LIN {X 0,Y 537.563,Z 430.245,A -85,B 0,C 180,E1 25559.467,E2 25559.467} C_VEL
LIN {X 0,Y 537.611,Z 430.26,A -85,B 0,C 180,E1 25556.268,E2 25556.268} C_VEL
LIN {X 0,Y 537.564,Z 430.265,A -85,B 0,C 180,E1 25552.948,E2 25552.948} C_VEL
LIN {X 0,Y 537.598,Z 430.246,A -85,B 0,C 180,E1 25549.606,E2 25549.606} C_VEL
LIN {X 0,Y 537.598,Z 430.246,A -85,B 0,C 180,E1 25546.337,E2 25546.337} C_VEL
LIN {X 0,Y 537.576,Z 430.262,A -85,B 0,C 180,E1 25542.949,E2 25542.949} C_VEL
LIN {X 0,Y 537.624,Z 430.26,A -85,B 0,C 180,E1 25539.613,E2 25539.613} C_VEL
LIN {X 0,Y 537.599,Z 430.262,A -85,B 0,C 180,E1 25536.313,E2 25536.313} C_VEL
LIN {X 0,Y 537.589,Z 430.264,A -85,B 0,C 180,E1 25532.891,E2 25532.891} C_VEL
LIN {X 0,Y 537.63,Z 430.257,A -85,B 0,C 180,E1 25529.611,E2 25529.611} C_VEL
LIN {X 0,Y 537.595,Z 430.198,A -85,B 0,C 180,E1 25526.212,E2 25526.212} C_VEL
LIN {X 0,Y 537.597,Z 430.248,A -85,B 0,C 180,E1 25522.755,E2 25522.755} C_VEL
LIN {X 0,Y 537.67,Z 430.675,A -85,B 0,C 180,E1 25522.164,E2 25522.164} C_VEL
LIN {X 0,Y 539.489,Z 434.5,A -85,B 0,C 180,E1 25521.457,E2 25521.457} C_VEL
LIN {X 0,Y 545.731,Z 448.172,A -85,B 0,C 180,E1 25519.149,E2 25519.149} C_VEL
LIN {X 0,Y 551.276,Z 460.441,A -85,B 0,C 180,E1 25517.249,E2 25517.249} C_VEL
LIN {X 0,Y 565.395,Z 481.878,A -85,B 0,C 180,E1 25515.423,E2 25515.423} C_VEL
LIN {X 0,Y 579.093,Z 504.577,A -85,B 0,C 180,E1 25513.764,E2 25513.764} C_VEL
LIN {X 0,Y 572.062,Z 749.764,A -85,B 0,C 180,E1 25510.284,E2 25510.284} C_VEL
LIN {X 0,Y 569.354,Z 843.896,A -85,B 0,C 180,E1 25508.929,E2 25508.929} C_VEL
LIN {X 0,Y 567.836,Z 869.316,A -85,B 0,C 180,E1 25508.396,E2 25508.396} C_VEL
LIN {X 0,Y 566.137,Z 891.39,A -85,B 0,C 180,E1 25507.777,E2 25507.777} C_VEL
LIN {X 0,Y 563.86,Z 915.912,A -85,B 0,C 180,E1 25506.893,E2 25506.893} C_VEL
LIN {X 0,Y 561.758,Z 935.486,A -85,B 0,C 180,E1 25506.034,E2 25506.034} C_VEL
LIN {X 0,Y 559.066,Z 958.281,A -85,B 0,C 180,E1 25504.85,E2 25504.85} C_VEL
LIN {X 0,Y 556.415,Z 978.46,A -85,B 0,C 180,E1 25503.607,E2 25503.607} C_VEL
LIN {X 0,Y 553.585,Z 999.25,A -85,B 0,C 180,E1 25502.13,E2 25502.13} C_VEL
LIN {X 0,Y 550.795,Z 1018.62,A -85,B 0,C 180,E1 25500.52,E2 25500.52} C_VEL
LIN {X 0,Y 548.082,Z 1037.54,A -85,B 0,C 180,E1 25498.732,E2 25498.732} C_VEL
LIN {X 0,Y 545.584,Z 1054.652,A -85,B 0,C 180,E1 25496.857,E2 25496.857} C_VEL
LIN {X 0,Y 543.312,Z 1071.181,A -85,B 0,C 180,E1 25494.81,E2 25494.81} C_VEL
LIN {X 0,Y 541.344,Z 1085.798,A -85,B 0,C 180,E1 25492.708,E2 25492.708} C_VEL
LIN {X 0,Y 539.711,Z 1099.37,A -85,B 0,C 180,E1 25490.497,E2 25490.497} C_VEL
LIN {X 0,Y 538.397,Z 1111.524,A -85,B 0,C 180,E1 25488.18,E2 25488.18} C_VEL
LIN {X 0,Y 537.464,Z 1121.5,A -85,B 0,C 180,E1 25485.982,E2 25485.982} C_VEL
LIN {X 0,Y 536.711,Z 1131.437,A -85,B 0,C 180,E1 25483.357,E2 25483.357} C_VEL
LIN {X 0,Y 536.314,Z 1137.908,A -85,B 0,C 180,E1 25481.285,E2 25481.285} C_VEL
LIN {X 0,Y 536.061,Z 1144.005,A -85,B 0,C 180,E1 25478.906,E2 25478.906} C_VEL
LIN {X 0,Y 535.956,Z 1148.651,A -85,B 0,C 180,E1 25476.427,E2 25476.427} C_VEL
LIN {X 0,Y 535.926,Z 1151.599,A -85,B 0,C 180,E1 25474.173,E2 25474.173} C_VEL
LIN {X 0,Y 535.906,Z 1153.482,A -85,B 0,C 180,E1 25471.604,E2 25471.604} C_VEL
LIN {X 0,Y 535.895,Z 1153.67,A -85,B 0,C 180,E1 25469.252,E2 25469.252} C_VEL
LIN {X 0,Y 535.893,Z 1152.72,A -85,B 0,C 180,E1 25467.112,E2 25467.112} C_VEL
LIN {X 0,Y 535.911,Z 1150.294,A -85,B 0,C 180,E1 25464.647,E2 25464.647} C_VEL
LIN {X 0,Y 535.982,Z 1146.4,A -85,B 0,C 180,E1 25462.281,E2 25462.281} C_VEL
LIN {X 0,Y 536.155,Z 1141.661,A -85,B 0,C 180,E1 25460.121,E2 25460.121} C_VEL
LIN {X 0,Y 536.527,Z 1134.357,A -85,B 0,C 180,E1 25457.515,E2 25457.515} C_VEL
LIN {X 0,Y 537.075,Z 1126.302,A -85,B 0,C 180,E1 25455.223,E2 25455.223} C_VEL
LIN {X 0,Y 537.942,Z 1116.295,A -85,B 0,C 180,E1 25452.81,E2 25452.81} C_VEL
LIN {X 0,Y 539.101,Z 1104.77,A -85,B 0,C 180,E1 25450.497,E2 25450.497} C_VEL
LIN {X 0,Y 540.565,Z 1092.172,A -85,B 0,C 180,E1 25448.288,E2 25448.288} C_VEL
LIN {X 0,Y 542.432,Z 1077.521,A -85,B 0,C 180,E1 25446.075,E2 25446.075} C_VEL
LIN {X 0,Y 544.396,Z 1063.086,A -85,B 0,C 180,E1 25444.156,E2 25444.156} C_VEL
LIN {X 0,Y 547.004,Z 1044.796,A -85,B 0,C 180,E1 25442.039,E2 25442.039} C_VEL
LIN {X 0,Y 549.352,Z 1028.487,A -85,B 0,C 180,E1 25440.385,E2 25440.385} C_VEL
LIN {X 0,Y 552.424,Z 1007.258,A -85,B 0,C 180,E1 25438.515,E2 25438.515} C_VEL
LIN {X 0,Y 554.922,Z 989.488,A -85,B 0,C 180,E1 25437.155,E2 25437.155} C_VEL
LIN {X 0,Y 557.868,Z 967.473,A -85,B 0,C 180,E1 25435.695,E2 25435.695} C_VEL
LIN {X 0,Y 560.34,Z 947.273,A -85,B 0,C 180,E1 25434.553,E2 25434.553} C_VEL
LIN {X 0,Y 563.059,Z 923.705,A -85,B 0,C 180,E1 25433.431,E2 25433.431} C_VEL
LIN {X 0,Y 565.125,Z 902.488,A -85,B 0,C 180,E1 25432.602,E2 25432.602} C_VEL
LIN {X 0,Y 567.194,Z 878.756,A -85,B 0,C 180,E1 25431.848,E2 25431.848} C_VEL
LIN {X 0,Y 568.742,Z 855.353,A -85,B 0,C 180,E1 25431.295,E2 25431.295} C_VEL
LIN {X 0,Y 569.818,Z 831.659,A -85,B 0,C 180,E1 25430.878,E2 25430.878} C_VEL
LIN {X 0,Y 576.437,Z 593.145,A -85,B 0,C 180,E1 25427.493,E2 25427.493} C_VEL
LIN {X 0,Y 578.891,Z 504.261,A -85,B 0,C 180,E1 25426.219,E2 25426.219} C_VEL
LIN {X 0,Y 564.561,Z 480.573,A -85,B 0,C 180,E1 25424.483,E2 25424.483} C_VEL
LIN {X 0,Y 551.107,Z 460.145,A -85,B 0,C 180,E1 25422.732,E2 25422.732} C_VEL
LIN {X 0,Y 544.782,Z 446.05,A -85,B 0,C 180,E1 25420.521,E2 25420.521} C_VEL
LIN {X 0,Y 539.013,Z 433.83,A -85,B 0,C 180,E1 25418.421,E2 25418.421} C_VEL
LIN {X 0,Y 537.627,Z 430.435,A -85,B 0,C 180,E1 25417.774,E2 25417.774} C_VEL
LIN {X 0,Y 537.619,Z 430.197,A -85,B 0,C 180,E1 25414.43,E2 25414.43} C_VEL
LIN {X 0,Y 537.596,Z 430.267,A -85,B 0,C 180,E1 25411.135,E2 25411.135} C_VEL
LIN {X 0,Y 537.604,Z 430.267,A -85,B 0,C 180,E1 25407.709,E2 25407.709} C_VEL
LIN {X 0,Y 537.629,Z 430.259,A -85,B 0,C 180,E1 25404.312,E2 25404.312} C_VEL
LIN {X 0,Y 537.586,Z 430.261,A -85,B 0,C 180,E1 25400.98,E2 25400.98} C_VEL
LIN {X 0,Y 537.59,Z 430.25,A -85,B 0,C 180,E1 25397.536,E2 25397.536} C_VEL
LIN {X 0,Y 537.633,Z 430.239,A -85,B 0,C 180,E1 25394.211,E2 25394.211} C_VEL
LIN {X 0,Y 537.573,Z 430.257,A -85,B 0,C 180,E1 25390.86,E2 25390.86} C_VEL
LIN {X 0,Y 537.591,Z 430.266,A -85,B 0,C 180,E1 25387.481,E2 25387.481} C_VEL
LIN {X 0,Y 537.597,Z 430.253,A -85,B 0,C 180,E1 25384.267,E2 25384.267} C_VEL
LIN {X 0,Y 537.56,Z 430.244,A -85,B 0,C 180,E1 25380.959,E2 25380.959} C_VEL
LIN {X 0,Y 537.618,Z 430.255,A -85,B 0,C 180,E1 25377.762,E2 25377.762} C_VEL
LIN {X 0,Y 537.561,Z 430.266,A -85,B 0,C 180,E1 25374.449,E2 25374.449} C_VEL
LIN {X 0,Y 537.558,Z 430.254,A -85,B 0,C 180,E1 25371.003,E2 25371.003} C_VEL
LIN {X 0,Y 537.604,Z 430.244,A -85,B 0,C 180,E1 25367.759,E2 25367.759} C_VEL
LIN {X 0,Y 537.545,Z 430.267,A -85,B 0,C 180,E1 25364.574,E2 25364.574} C_VEL
LIN {X 0,Y 537.598,Z 430.266,A -85,B 0,C 180,E1 25361.343,E2 25361.343} C_VEL
LIN {X 0,Y 537.544,Z 430.262,A -85,B 0,C 180,E1 25358.156,E2 25358.156} C_VEL
LIN {X 0,Y 537.539,Z 430.259,A -85,B 0,C 180,E1 25354.67,E2 25354.67} C_VEL
LIN {X 0,Y 537.604,Z 430.249,A -85,B 0,C 180,E1 25351.387,E2 25351.387} C_VEL
LIN {X 0,Y 537.524,Z 430.258,A -85,B 0,C 180,E1 25348.223,E2 25348.223} C_VEL
LIN {X 0,Y 537.558,Z 430.212,A -85,B 0,C 180,E1 25344.917,E2 25344.917} C_VEL
LIN {X 0,Y 537.544,Z 430.254,A -85,B 0,C 180,E1 25341.718,E2 25341.718} C_VEL
LIN {X 0,Y 537.659,Z 430.659,A -85,B 0,C 180,E1 25341.25,E2 25341.25} C_VEL
LIN {X 0,Y 539.072,Z 434.068,A -85,B 0,C 180,E1 25340.628,E2 25340.628} C_VEL
LIN {X 0,Y 543.735,Z 444.332,A -85,B 0,C 180,E1 25338.827,E2 25338.827} C_VEL
LIN {X 0,Y 548.585,Z 455.234,A -85,B 0,C 180,E1 25337.025,E2 25337.025} C_VEL
LIN {X 0,Y 555.423,Z 471.599,A -85,B 0,C 180,E1 25334.529,E2 25334.529} C_VEL
LIN {X 0,Y 562.151,Z 489.574,A -85,B 0,C 180,E1 25332.046,E2 25332.046} C_VEL
LIN {X 0,Y 563.644,Z 493.192,A -85,B 0,C 180,E1 25331.625,E2 25331.625} C_VEL
LIN {X 0,Y 567.174,Z 499.748,A -85,B 0,C 180,E1 25331.178,E2 25331.178} C_VEL
LIN {X 0,Y 575.924,Z 543.536,A -85,B 0,C 180,E1 25329.673,E2 25329.673} C_VEL
LIN {X 0,Y 570.099,Z 791.217,A -85,B 0,C 180,E1 25326.365,E2 25326.365} C_VEL
LIN {X 0,Y 569.15,Z 798.915,A -85,B 0,C 180,E1 25326.325,E2 25326.325} C_VEL
LIN {X 0,Y 563.752,Z 819.438,A -85,B 0,C 180,E1 25326.446,E2 25326.446} C_VEL
LIN {X 0,Y 563.016,Z 826.045,A -85,B 0,C 180,E1 25326.405,E2 25326.405} C_VEL
LIN {X 0,Y 561.954,Z 855.614,A -85,B 0,C 180,E1 25325.948,E2 25325.948} C_VEL
LIN {X 0,Y 560.633,Z 876.398,A -85,B 0,C 180,E1 25325.48,E2 25325.48} C_VEL
LIN {X 0,Y 558.691,Z 899.351,A -85,B 0,C 180,E1 25324.782,E2 25324.782} C_VEL
LIN {X 0,Y 556.656,Z 919.096,A -85,B 0,C 180,E1 25324.024,E2 25324.024} C_VEL
LIN {X 0,Y 553.94,Z 941.342,A -85,B 0,C 180,E1 25322.972,E2 25322.972} C_VEL
LIN {X 0,Y 551.282,Z 960.921,A -85,B 0,C 180,E1 25321.857,E2 25321.857} C_VEL
LIN {X 0,Y 548.337,Z 980.641,A -85,B 0,C 180,E1 25320.521,E2 25320.521} C_VEL
LIN {X 0,Y 545.53,Z 998.333,A -85,B 0,C 180,E1 25319.127,E2 25319.127} C_VEL
LIN {X 0,Y 542.444,Z 1016.652,A -85,B 0,C 180,E1 25317.441,E2 25317.441} C_VEL
LIN {X 0,Y 539.637,Z 1033.467,A -85,B 0,C 180,E1 25315.651,E2 25315.651} C_VEL
LIN {X 0,Y 536.965,Z 1048.953,A -85,B 0,C 180,E1 25313.717,E2 25313.717} C_VEL
LIN {X 0,Y 534.607,Z 1063.539,A -85,B 0,C 180,E1 25311.62,E2 25311.62} C_VEL
LIN {X 0,Y 532.672,Z 1075.997,A -85,B 0,C 180,E1 25309.52,E2 25309.52} C_VEL
LIN {X 0,Y 530.943,Z 1088.34,A -85,B 0,C 180,E1 25307.085,E2 25307.085} C_VEL
LIN {X 0,Y 529.803,Z 1097.772,A -85,B 0,C 180,E1 25304.873,E2 25304.873} C_VEL
LIN {X 0,Y 528.907,Z 1106.716,A -85,B 0,C 180,E1 25302.335,E2 25302.335} C_VEL
LIN {X 0,Y 528.402,Z 1113.315,A -85,B 0,C 180,E1 25300.026,E2 25300.026} C_VEL
LIN {X 0,Y 528.103,Z 1118.824,A -85,B 0,C 180,E1 25297.507,E2 25297.507} C_VEL
LIN {X 0,Y 527.976,Z 1122.478,A -85,B 0,C 180,E1 25295.216,E2 25295.216} C_VEL
LIN {X 0,Y 527.922,Z 1124.991,A -85,B 0,C 180,E1 25292.605,E2 25292.605} C_VEL
LIN {X 0,Y 527.918,Z 1125.857,A -85,B 0,C 180,E1 25290.326,E2 25290.326} C_VEL
LIN {X 0,Y 527.922,Z 1125.244,A -85,B 0,C 180,E1 25287.72,E2 25287.72} C_VEL
LIN {X 0,Y 527.946,Z 1123.366,A -85,B 0,C 180,E1 25285.438,E2 25285.438} C_VEL
LIN {X 0,Y 528.064,Z 1119.589,A -85,B 0,C 180,E1 25282.821,E2 25282.821} C_VEL
LIN {X 0,Y 528.304,Z 1114.866,A -85,B 0,C 180,E1 25280.522,E2 25280.522} C_VEL
LIN {X 0,Y 528.798,Z 1108.023,A -85,B 0,C 180,E1 25277.995,E2 25277.995} C_VEL
LIN {X 0,Y 529.546,Z 1100.239,A -85,B 0,C 180,E1 25275.679,E2 25275.679} C_VEL
LIN {X 0,Y 530.706,Z 1090.239,A -85,B 0,C 180,E1 25273.246,E2 25273.246} C_VEL
LIN {X 0,Y 532.27,Z 1078.959,A -85,B 0,C 180,E1 25270.921,E2 25270.921} C_VEL
LIN {X 0,Y 534.178,Z 1066.132,A -85,B 0,C 180,E1 25268.707,E2 25268.707} C_VEL
LIN {X 0,Y 536.604,Z 1051.259,A -85,B 0,C 180,E1 25266.499,E2 25266.499} C_VEL
LIN {X 0,Y 539.08,Z 1036.58,A -85,B 0,C 180,E1 25264.63,E2 25264.63} C_VEL
LIN {X 0,Y 542.044,Z 1019.136,A -85,B 0,C 180,E1 25262.716,E2 25262.716} C_VEL
LIN {X 0,Y 544.839,Z 1002.518,A -85,B 0,C 180,E1 25261.141,E2 25261.141} C_VEL
LIN {X 0,Y 547.91,Z 983.484,A -85,B 0,C 180,E1 25259.597,E2 25259.597} C_VEL
LIN {X 0,Y 550.709,Z 965.137,A -85,B 0,C 180,E1 25258.317,E2 25258.317} C_VEL
LIN {X 0,Y 553.497,Z 944.852,A -85,B 0,C 180,E1 25257.122,E2 25257.122} C_VEL
LIN {X 0,Y 556.047,Z 924.615,A -85,B 0,C 180,E1 25256.12,E2 25256.12} C_VEL
LIN {X 0,Y 558.333,Z 903.1,A -85,B 0,C 180,E1 25255.256,E2 25255.256} C_VEL
LIN {X 0,Y 560.263,Z 881.795,A -85,B 0,C 180,E1 25254.571,E2 25254.571} C_VEL
LIN {X 0,Y 561.795,Z 858.909,A -85,B 0,C 180,E1 25254.024,E2 25254.024} C_VEL
LIN {X 0,Y 562.808,Z 836.018,A -85,B 0,C 180,E1 25253.636,E2 25253.636} C_VEL
LIN {X 0,Y 568.803,Z 586.916,A -85,B 0,C 180,E1 25250.287,E2 25250.287} C_VEL
LIN {X 0,Y 569.81,Z 544.081,A -85,B 0,C 180,E1 25249.691,E2 25249.691} C_VEL
LIN {X 0,Y 561.524,Z 502.952,A -85,B 0,C 180,E1 25248.235,E2 25248.235} C_VEL
LIN {X 0,Y 554.808,Z 491.423,A -85,B 0,C 180,E1 25247.334,E2 25247.334} C_VEL
LIN {X 0,Y 547.67,Z 472.631,A -85,B 0,C 180,E1 25244.66,E2 25244.66} C_VEL
LIN {X 0,Y 540.405,Z 455.19,A -85,B 0,C 180,E1 25241.909,E2 25241.909} C_VEL
LIN {X 0,Y 534.741,Z 442.856,A -85,B 0,C 180,E1 25239.754,E2 25239.754} C_VEL
LIN {X 0,Y 531.038,Z 434.894,A -85,B 0,C 180,E1 25238.278,E2 25238.278} C_VEL
LIN {X 0,Y 529.624,Z 431.422,A -85,B 0,C 180,E1 25237.575,E2 25237.575} C_VEL
LIN {X 0,Y 529.637,Z 431.208,A -85,B 0,C 180,E1 25234.497,E2 25234.497} C_VEL
LIN {X 0,Y 529.602,Z 431.244,A -85,B 0,C 180,E1 25231.279,E2 25231.279} C_VEL
LIN {X 0,Y 529.59,Z 431.245,A -85,B 0,C 180,E1 25227.919,E2 25227.919} C_VEL
LIN {X 0,Y 529.649,Z 431.237,A -85,B 0,C 180,E1 25224.659,E2 25224.659} C_VEL
LIN {X 0,Y 529.592,Z 431.247,A -85,B 0,C 180,E1 25221.439,E2 25221.439} C_VEL
LIN {X 0,Y 529.637,Z 431.25,A -85,B 0,C 180,E1 25218.15,E2 25218.15} C_VEL
LIN {X 0,Y 529.613,Z 431.258,A -85,B 0,C 180,E1 25214.99,E2 25214.99} C_VEL
LIN {X 0,Y 529.607,Z 431.248,A -85,B 0,C 180,E1 25211.516,E2 25211.516} C_VEL
LIN {X 0,Y 529.676,Z 431.228,A -85,B 0,C 180,E1 25208.249,E2 25208.249} C_VEL
LIN {X 0,Y 529.617,Z 431.251,A -85,B 0,C 180,E1 25204.982,E2 25204.982} C_VEL
LIN {X 0,Y 529.625,Z 431.257,A -85,B 0,C 180,E1 25201.515,E2 25201.515} C_VEL
LIN {X 0,Y 529.662,Z 431.233,A -85,B 0,C 180,E1 25198.377,E2 25198.377} C_VEL
LIN {X 0,Y 529.621,Z 431.237,A -85,B 0,C 180,E1 25195.018,E2 25195.018} C_VEL
LIN {X 0,Y 529.661,Z 431.248,A -85,B 0,C 180,E1 25191.642,E2 25191.642} C_VEL
LIN {X 0,Y 529.66,Z 431.251,A -85,B 0,C 180,E1 25188.346,E2 25188.346} C_VEL
LIN {X 0,Y 529.634,Z 431.241,A -85,B 0,C 180,E1 25185.01,E2 25185.01} C_VEL
LIN {X 0,Y 529.685,Z 431.228,A -85,B 0,C 180,E1 25181.718,E2 25181.718} C_VEL
LIN {X 0,Y 529.653,Z 431.237,A -85,B 0,C 180,E1 25178.4,E2 25178.4} C_VEL
LIN {X 0,Y 529.651,Z 431.243,A -85,B 0,C 180,E1 25174.98,E2 25174.98} C_VEL
LIN {X 0,Y 529.696,Z 431.238,A -85,B 0,C 180,E1 25171.595,E2 25171.595} C_VEL
LIN {X 0,Y 529.663,Z 431.229,A -85,B 0,C 180,E1 25168.218,E2 25168.218} C_VEL
LIN {X 0,Y 529.65,Z 431.203,A -85,B 0,C 180,E1 25164.712,E2 25164.712} C_VEL
LIN {X 0,Y 529.728,Z 431.569,A -85,B 0,C 180,E1 25163.161,E2 25163.161} C_VEL
LIN {X 0,Y 531.079,Z 434.887,A -85,B 0,C 180,E1 25162.545,E2 25162.545} C_VEL
LIN {X 0,Y 534.312,Z 441.615,A -85,B 0,C 180,E1 25161.315,E2 25161.315} C_VEL
LIN {X 0,Y 539.492,Z 452.574,A -85,B 0,C 180,E1 25159.417,E2 25159.417} C_VEL
LIN {X 0,Y 543.297,Z 460.954,A -85,B 0,C 180,E1 25158.099,E2 25158.099} C_VEL
LIN {X 0,Y 557.37,Z 482.066,A -85,B 0,C 180,E1 25156.21,E2 25156.21} C_VEL
LIN {X 0,Y 571.534,Z 505.199,A -85,B 0,C 180,E1 25154.438,E2 25154.438} C_VEL
LIN {X 0,Y 573.043,Z 508.177,A -85,B 0,C 180,E1 25154.248,E2 25154.248} C_VEL
LIN {X 0,Y 565.685,Z 754.075,A -85,B 0,C 180,E1 25150.727,E2 25150.727} C_VEL
LIN {X 0,Y 562.975,Z 844.037,A -85,B 0,C 180,E1 25149.419,E2 25149.419} C_VEL
LIN {X 0,Y 561.402,Z 869.3,A -85,B 0,C 180,E1 25148.885,E2 25148.885} C_VEL
LIN {X 0,Y 559.62,Z 891.562,A -85,B 0,C 180,E1 25148.255,E2 25148.255} C_VEL
LIN {X 0,Y 557.329,Z 915.295,A -85,B 0,C 180,E1 25147.394,E2 25147.394} C_VEL
LIN {X 0,Y 555.015,Z 935.997,A -85,B 0,C 180,E1 25146.478,E2 25146.478} C_VEL
LIN {X 0,Y 552.089,Z 959.513,A -85,B 0,C 180,E1 25145.233,E2 25145.233} C_VEL
LIN {X 0,Y 549.449,Z 978.788,A -85,B 0,C 180,E1 25144.028,E2 25144.028} C_VEL
LIN {X 0,Y 546.495,Z 999.423,A -85,B 0,C 180,E1 25142.542,E2 25142.542} C_VEL
LIN {X 0,Y 543.614,Z 1018.503,A -85,B 0,C 180,E1 25140.937,E2 25140.937} C_VEL
LIN {X 0,Y 540.813,Z 1037.151,A -85,B 0,C 180,E1 25139.155,E2 25139.155} C_VEL
LIN {X 0,Y 538.096,Z 1054.746,A -85,B 0,C 180,E1 25137.201,E2 25137.201} C_VEL
LIN {X 0,Y 535.733,Z 1071.067,A -85,B 0,C 180,E1 25135.149,E2 25135.149} C_VEL
LIN {X 0,Y 533.588,Z 1086.161,A -85,B 0,C 180,E1 25132.94,E2 25132.94} C_VEL
LIN {X 0,Y 531.882,Z 1099.66,A -85,B 0,C 180,E1 25130.697,E2 25130.697} C_VEL
LIN {X 0,Y 530.496,Z 1111.691,A -85,B 0,C 180,E1 25128.347,E2 25128.347} C_VEL
LIN {X 0,Y 529.483,Z 1122.099,A -85,B 0,C 180,E1 25126.004,E2 25126.004} C_VEL
LIN {X 0,Y 528.734,Z 1131.506,A -85,B 0,C 180,E1 25123.451,E2 25123.451} C_VEL
LIN {X 0,Y 528.31,Z 1138.247,A -85,B 0,C 180,E1 25121.241,E2 25121.241} C_VEL
LIN {X 0,Y 528.052,Z 1144.655,A -85,B 0,C 180,E1 25118.603,E2 25118.603} C_VEL
LIN {X 0,Y 527.955,Z 1148.75,A -85,B 0,C 180,E1 25116.306,E2 25116.306} C_VEL
LIN {X 0,Y 527.925,Z 1151.615,A -85,B 0,C 180,E1 25114.018,E2 25114.018} C_VEL
LIN {X 0,Y 527.916,Z 1153.342,A -85,B 0,C 180,E1 25111.302,E2 25111.302} C_VEL
LIN {X 0,Y 527.902,Z 1153.437,A -85,B 0,C 180,E1 25109.132,E2 25109.132} C_VEL
LIN {X 0,Y 527.899,Z 1152.434,A -85,B 0,C 180,E1 25106.96,E2 25106.96} C_VEL
LIN {X 0,Y 527.927,Z 1149.742,A -85,B 0,C 180,E1 25104.348,E2 25104.348} C_VEL
LIN {X 0,Y 528,Z 1145.941,A -85,B 0,C 180,E1 25102.054,E2 25102.054} C_VEL
LIN {X 0,Y 528.189,Z 1140.872,A -85,B 0,C 180,E1 25099.75,E2 25099.75} C_VEL
LIN {X 0,Y 528.611,Z 1133.332,A -85,B 0,C 180,E1 25097.103,E2 25097.103} C_VEL
LIN {X 0,Y 529.183,Z 1125.554,A -85,B 0,C 180,E1 25094.885,E2 25094.885} C_VEL
LIN {X 0,Y 530.17,Z 1114.882,A -85,B 0,C 180,E1 25092.323,E2 25092.323} C_VEL
LIN {X 0,Y 531.368,Z 1103.818,A -85,B 0,C 180,E1 25090.087,E2 25090.087} C_VEL
LIN {X 0,Y 533.053,Z 1090.481,A -85,B 0,C 180,E1 25087.734,E2 25087.734} C_VEL
LIN {X 0,Y 535.015,Z 1075.841,A -85,B 0,C 180,E1 25085.527,E2 25085.527} C_VEL
LIN {X 0,Y 537.29,Z 1060.404,A -85,B 0,C 180,E1 25083.472,E2 25083.472} C_VEL
LIN {X 0,Y 539.885,Z 1042.843,A -85,B 0,C 180,E1 25081.456,E2 25081.456} C_VEL
LIN {X 0,Y 542.709,Z 1024.671,A -85,B 0,C 180,E1 25079.619,E2 25079.619} C_VEL
LIN {X 0,Y 545.521,Z 1005.807,A -85,B 0,C 180,E1 25077.979,E2 25077.979} C_VEL
LIN {X 0,Y 548.322,Z 986.768,A -85,B 0,C 180,E1 25076.521,E2 25076.521} C_VEL
LIN {X 0,Y 551.332,Z 964.918,A -85,B 0,C 180,E1 25075.091,E2 25075.091} C_VEL
LIN {X 0,Y 553.941,Z 944.652,A -85,B 0,C 180,E1 25073.953,E2 25073.953} C_VEL
LIN {X 0,Y 556.71,Z 921.019,A -85,B 0,C 180,E1 25072.847,E2 25072.847} C_VEL
LIN {X 0,Y 558.801,Z 900.349,A -85,B 0,C 180,E1 25072.046,E2 25072.046} C_VEL
LIN {X 0,Y 560.965,Z 875.428,A -85,B 0,C 180,E1 25071.276,E2 25071.276} C_VEL
LIN {X 0,Y 562.43,Z 853.769,A -85,B 0,C 180,E1 25070.772,E2 25070.772} C_VEL
LIN {X 0,Y 563.576,Z 827.693,A -85,B 0,C 180,E1 25070.327,E2 25070.327} C_VEL
LIN {X 0,Y 570.432,Z 591.297,A -85,B 0,C 180,E1 25066.942,E2 25066.942} C_VEL
LIN {X 0,Y 572.854,Z 507.561,A -85,B 0,C 180,E1 25065.731,E2 25065.731} C_VEL
LIN {X 0,Y 559.284,Z 485.093,A -85,B 0,C 180,E1 25064.046,E2 25064.046} C_VEL
LIN {X 0,Y 545.384,Z 464.099,A -85,B 0,C 180,E1 25062.216,E2 25062.216} C_VEL
LIN {X 0,Y 542.908,Z 460.138,A -85,B 0,C 180,E1 25061.814,E2 25061.814} C_VEL
LIN {X 0,Y 535.54,Z 443.92,A -85,B 0,C 180,E1 25059.129,E2 25059.129} C_VEL
LIN {X 0,Y 531.026,Z 434.81,A -85,B 0,C 180,E1 25057.459,E2 25057.459} C_VEL
LIN {X 0,Y 529.703,Z 431.4,A -85,B 0,C 180,E1 25056.796,E2 25056.796} C_VEL
LIN {X 0,Y 529.647,Z 431.187,A -85,B 0,C 180,E1 25053.443,E2 25053.443} C_VEL
LIN {X 0,Y 529.685,Z 431.239,A -85,B 0,C 180,E1 25050.016,E2 25050.016} C_VEL
LIN {X 0,Y 529.683,Z 431.239,A -85,B 0,C 180,E1 25046.576,E2 25046.576} C_VEL
LIN {X 0,Y 529.645,Z 431.246,A -85,B 0,C 180,E1 25043.163,E2 25043.163} C_VEL
LIN {X 0,Y 529.67,Z 431.247,A -85,B 0,C 180,E1 25039.75,E2 25039.75} C_VEL
LIN {X 0,Y 529.682,Z 431.249,A -85,B 0,C 180,E1 25036.336,E2 25036.336} C_VEL
LIN {X 0,Y 529.633,Z 431.247,A -85,B 0,C 180,E1 25033.054,E2 25033.054} C_VEL
LIN {X 0,Y 529.666,Z 431.231,A -85,B 0,C 180,E1 25029.672,E2 25029.672} C_VEL
LIN {X 0,Y 529.645,Z 431.245,A -85,B 0,C 180,E1 25026.504,E2 25026.504} C_VEL
LIN {X 0,Y 529.627,Z 431.257,A -85,B 0,C 180,E1 25023.03,E2 25023.03} C_VEL
LIN {X 0,Y 529.678,Z 431.237,A -85,B 0,C 180,E1 25019.676,E2 25019.676} C_VEL
LIN {X 0,Y 529.625,Z 431.232,A -85,B 0,C 180,E1 25016.428,E2 25016.428} C_VEL
LIN {X 0,Y 529.618,Z 431.247,A -85,B 0,C 180,E1 25012.951,E2 25012.951} C_VEL
LIN {X 0,Y 529.675,Z 431.253,A -85,B 0,C 180,E1 25009.669,E2 25009.669} C_VEL
LIN {X 0,Y 529.612,Z 431.249,A -85,B 0,C 180,E1 25006.35,E2 25006.35} C_VEL
LIN {X 0,Y 529.609,Z 431.24,A -85,B 0,C 180,E1 25002.809,E2 25002.809} C_VEL
LIN {X 0,Y 529.664,Z 431.235,A -85,B 0,C 180,E1 24999.559,E2 24999.559} C_VEL
LIN {X 0,Y 529.598,Z 431.252,A -85,B 0,C 180,E1 24996.305,E2 24996.305} C_VEL
LIN {X 0,Y 529.62,Z 431.253,A -85,B 0,C 180,E1 24992.935,E2 24992.935} C_VEL
LIN {X 0,Y 529.609,Z 431.262,A -85,B 0,C 180,E1 24989.848,E2 24989.848} C_VEL
LIN {X 0,Y 529.587,Z 431.253,A -85,B 0,C 180,E1 24986.413,E2 24986.413} C_VEL
LIN {X 0,Y 529.644,Z 431.193,A -85,B 0,C 180,E1 24983.106,E2 24983.106} C_VEL
LIN {X 0,Y 529.642,Z 431.592,A -85,B 0,C 180,E1 24982.243,E2 24982.243} C_VEL
LIN {X 0,Y 531.101,Z 434.984,A -85,B 0,C 180,E1 24981.59,E2 24981.59} C_VEL
LIN {X 0,Y 537.213,Z 447.995,A -85,B 0,C 180,E1 24979.209,E2 24979.209} C_VEL
LIN {X 0,Y 544.385,Z 464.616,A -85,B 0,C 180,E1 24976.466,E2 24976.466} C_VEL
LIN {X 0,Y 551.341,Z 482.15,A -85,B 0,C 180,E1 24973.851,E2 24973.851} C_VEL
LIN {X 0,Y 555.2,Z 492.369,A -85,B 0,C 180,E1 24972.475,E2 24972.475} C_VEL
LIN {X 0,Y 561.756,Z 503.833,A -85,B 0,C 180,E1 24971.629,E2 24971.629} C_VEL
LIN {X 0,Y 569.904,Z 545.198,A -85,B 0,C 180,E1 24970.185,E2 24970.185} C_VEL
LIN {X 0,Y 563.405,Z 809.503,A -85,B 0,C 180,E1 24966.625,E2 24966.625} C_VEL
LIN {X 0,Y 563.016,Z 826.045,A -85,B 0,C 180,E1 24966.405,E2 24966.405} C_VEL
LIN {X 0,Y 562.045,Z 833.733,A -85,B 0,C 180,E1 24966.367,E2 24966.367} C_VEL
LIN {X 0,Y 556.549,Z 853.082,A -85,B 0,C 180,E1 24966.445,E2 24966.445} C_VEL
LIN {X 0,Y 555.344,Z 860.705,A -85,B 0,C 180,E1 24966.354,E2 24966.354} C_VEL
LIN {X 0,Y 553.548,Z 885.065,A -85,B 0,C 180,E1 24965.741,E2 24965.741} C_VEL
LIN {X 0,Y 551.55,Z 906.159,A -85,B 0,C 180,E1 24965.039,E2 24965.039} C_VEL
LIN {X 0,Y 549.048,Z 927.998,A -85,B 0,C 180,E1 24964.119,E2 24964.119} C_VEL
LIN {X 0,Y 546.406,Z 948.141,A -85,B 0,C 180,E1 24963.092,E2 24963.092} C_VEL
LIN {X 0,Y 543.351,Z 968.81,A -85,B 0,C 180,E1 24961.818,E2 24961.818} C_VEL
LIN {X 0,Y 540.368,Z 987.586,A -85,B 0,C 180,E1 24960.465,E2 24960.465} C_VEL
LIN {X 0,Y 537.166,Z 1006.152,A -85,B 0,C 180,E1 24958.884,E2 24958.884} C_VEL
LIN {X 0,Y 534.154,Z 1023.522,A -85,B 0,C 180,E1 24957.178,E2 24957.178} C_VEL
LIN {X 0,Y 531.194,Z 1039.825,A -85,B 0,C 180,E1 24955.296,E2 24955.296} C_VEL
LIN {X 0,Y 528.426,Z 1055.683,A -85,B 0,C 180,E1 24953.178,E2 24953.178} C_VEL
LIN {X 0,Y 526.221,Z 1068.621,A -85,B 0,C 180,E1 24951.163,E2 24951.163} C_VEL
LIN {X 0,Y 524.178,Z 1081.598,A -85,B 0,C 180,E1 24948.807,E2 24948.807} C_VEL
LIN {X 0,Y 522.708,Z 1092.114,A -85,B 0,C 180,E1 24946.56,E2 24946.56} C_VEL
LIN {X 0,Y 521.53,Z 1101.75,A -85,B 0,C 180,E1 24944.093,E2 24944.093} C_VEL
LIN {X 0,Y 520.756,Z 1109.704,A -85,B 0,C 180,E1 24941.631,E2 24941.631} C_VEL
LIN {X 0,Y 520.285,Z 1115.884,A -85,B 0,C 180,E1 24939.179,E2 24939.179} C_VEL
LIN {X 0,Y 520.051,Z 1120.651,A -85,B 0,C 180,E1 24936.735,E2 24936.735} C_VEL
LIN {X 0,Y 519.952,Z 1123.929,A -85,B 0,C 180,E1 24934.191,E2 24934.191} C_VEL
LIN {X 0,Y 519.923,Z 1125.73,A -85,B 0,C 180,E1 24931.763,E2 24931.763} C_VEL
LIN {X 0,Y 519.919,Z 1125.997,A -85,B 0,C 180,E1 24929.229,E2 24929.229} C_VEL
LIN {X 0,Y 519.938,Z 1124.931,A -85,B 0,C 180,E1 24926.803,E2 24926.803} C_VEL
LIN {X 0,Y 519.993,Z 1122.21,A -85,B 0,C 180,E1 24924.261,E2 24924.261} C_VEL
LIN {X 0,Y 520.152,Z 1118.337,A -85,B 0,C 180,E1 24921.887,E2 24921.887} C_VEL
LIN {X 0,Y 520.508,Z 1112.623,A -85,B 0,C 180,E1 24919.373,E2 24919.373} C_VEL
LIN {X 0,Y 521.102,Z 1105.878,A -85,B 0,C 180,E1 24917.026,E2 24917.026} C_VEL
LIN {X 0,Y 522.068,Z 1097.059,A -85,B 0,C 180,E1 24914.56,E2 24914.56} C_VEL
LIN {X 0,Y 523.41,Z 1087.01,A -85,B 0,C 180,E1 24912.202,E2 24912.202} C_VEL
LIN {X 0,Y 525.108,Z 1075.543,A -85,B 0,C 180,E1 24909.955,E2 24909.955} C_VEL
LIN {X 0,Y 527.295,Z 1062.376,A -85,B 0,C 180,E1 24907.726,E2 24907.726} C_VEL
LIN {X 0,Y 529.708,Z 1048.274,A -85,B 0,C 180,E1 24905.701,E2 24905.701} C_VEL
LIN {X 0,Y 532.583,Z 1032.236,A -85,B 0,C 180,E1 24903.7,E2 24903.7} C_VEL
LIN {X 0,Y 535.415,Z 1016.232,A -85,B 0,C 180,E1 24901.986,E2 24901.986} C_VEL
LIN {X 0,Y 538.743,Z 997.221,A -85,B 0,C 180,E1 24900.233,E2 24900.233} C_VEL
LIN {X 0,Y 541.596,Z 980.023,A -85,B 0,C 180,E1 24898.873,E2 24898.873} C_VEL
LIN {X 0,Y 544.804,Z 959.229,A -85,B 0,C 180,E1 24897.469,E2 24897.469} C_VEL
LIN {X 0,Y 547.515,Z 940.119,A -85,B 0,C 180,E1 24896.384,E2 24896.384} C_VEL
LIN {X 0,Y 550.296,Z 917.88,A -85,B 0,C 180,E1 24895.339,E2 24895.339} C_VEL
LIN {X 0,Y 552.347,Z 898.644,A -85,B 0,C 180,E1 24894.6,E2 24894.6} C_VEL
LIN {X 0,Y 554.416,Z 874.565,A -85,B 0,C 180,E1 24893.876,E2 24893.876} C_VEL
LIN {X 0,Y 555.808,Z 853.164,A -85,B 0,C 180,E1 24893.402,E2 24893.402} C_VEL
LIN {X 0,Y 556.909,Z 820.613,A -85,B 0,C 180,E1 24892.918,E2 24892.918} C_VEL
LIN {X 0,Y 563.577,Z 560.669,A -85,B 0,C 180,E1 24889.388,E2 24889.388} C_VEL
LIN {X 0,Y 563.823,Z 545.677,A -85,B 0,C 180,E1 24889.164,E2 24889.164} C_VEL
LIN {X 0,Y 556.213,Z 507.334,A -85,B 0,C 180,E1 24887.787,E2 24887.787} C_VEL
LIN {X 0,Y 546.683,Z 491.01,A -85,B 0,C 180,E1 24886.486,E2 24886.486} C_VEL
LIN {X 0,Y 539.764,Z 473.202,A -85,B 0,C 180,E1 24883.854,E2 24883.854} C_VEL
LIN {X 0,Y 532.588,Z 456.293,A -85,B 0,C 180,E1 24881.079,E2 24881.079} C_VEL
LIN {X 0,Y 527.078,Z 444.218,A -85,B 0,C 180,E1 24878.897,E2 24878.897} C_VEL
LIN {X 0,Y 525.082,Z 440.053,A -85,B 0,C 180,E1 24878.096,E2 24878.096} C_VEL
LIN {X 0,Y 522.839,Z 435.45,A -85,B 0,C 180,E1 24877.181,E2 24877.181} C_VEL
LIN {X 0,Y 521.729,Z 432.388,A -85,B 0,C 180,E1 24876.548,E2 24876.548} C_VEL
LIN {X 0,Y 521.665,Z 432.243,A -85,B 0,C 180,E1 24873.374,E2 24873.374} C_VEL
LIN {X 0,Y 521.656,Z 432.253,A -85,B 0,C 180,E1 24869.892,E2 24869.892} C_VEL
LIN {X 0,Y 521.711,Z 432.244,A -85,B 0,C 180,E1 24866.646,E2 24866.646} C_VEL
LIN {X 0,Y 521.656,Z 432.247,A -85,B 0,C 180,E1 24863.345,E2 24863.345} C_VEL
LIN {X 0,Y 521.666,Z 432.238,A -85,B 0,C 180,E1 24859.832,E2 24859.832} C_VEL
LIN {X 0,Y 521.711,Z 432.222,A -85,B 0,C 180,E1 24856.593,E2 24856.593} C_VEL
LIN {X 0,Y 521.661,Z 432.235,A -85,B 0,C 180,E1 24853.411,E2 24853.411} C_VEL
LIN {X 0,Y 521.71,Z 432.242,A -85,B 0,C 180,E1 24850.044,E2 24850.044} C_VEL
LIN {X 0,Y 521.684,Z 432.236,A -85,B 0,C 180,E1 24846.825,E2 24846.825} C_VEL
LIN {X 0,Y 521.676,Z 432.222,A -85,B 0,C 180,E1 24843.406,E2 24843.406} C_VEL
LIN {X 0,Y 521.75,Z 432.221,A -85,B 0,C 180,E1 24840.11,E2 24840.11} C_VEL
LIN {X 0,Y 521.696,Z 432.247,A -85,B 0,C 180,E1 24836.704,E2 24836.704} C_VEL
LIN {X 0,Y 521.692,Z 432.239,A -85,B 0,C 180,E1 24833.286,E2 24833.286} C_VEL
LIN {X 0,Y 521.743,Z 432.217,A -85,B 0,C 180,E1 24829.956,E2 24829.956} C_VEL
LIN {X 0,Y 521.701,Z 432.228,A -85,B 0,C 180,E1 24826.591,E2 24826.591} C_VEL
LIN {X 0,Y 521.702,Z 432.24,A -85,B 0,C 180,E1 24823.063,E2 24823.063} C_VEL
LIN {X 0,Y 521.749,Z 432.238,A -85,B 0,C 180,E1 24819.704,E2 24819.704} C_VEL
LIN {X 0,Y 521.719,Z 432.239,A -85,B 0,C 180,E1 24816.363,E2 24816.363} C_VEL
LIN {X 0,Y 521.711,Z 432.242,A -85,B 0,C 180,E1 24812.861,E2 24812.861} C_VEL
LIN {X 0,Y 521.753,Z 432.237,A -85,B 0,C 180,E1 24809.479,E2 24809.479} C_VEL
LIN {X 0,Y 521.732,Z 432.168,A -85,B 0,C 180,E1 24805.971,E2 24805.971} C_VEL
LIN {X 0,Y 521.763,Z 432.501,A -85,B 0,C 180,E1 24804.21,E2 24804.21} C_VEL
LIN {X 0,Y 523.207,Z 435.938,A -85,B 0,C 180,E1 24803.534,E2 24803.534} C_VEL
LIN {X 0,Y 528.183,Z 446.106,A -85,B 0,C 180,E1 24801.604,E2 24801.604} C_VEL
LIN {X 0,Y 533.809,Z 458.448,A -85,B 0,C 180,E1 24799.46,E2 24799.46} C_VEL
LIN {X 0,Y 535.463,Z 461.704,A -85,B 0,C 180,E1 24798.964,E2 24798.964} C_VEL
LIN {X 0,Y 549.974,Z 483.29,A -85,B 0,C 180,E1 24796.946,E2 24796.946} C_VEL
LIN {X 0,Y 562.546,Z 503.462,A -85,B 0,C 180,E1 24795.316,E2 24795.316} C_VEL
LIN {X 0,Y 567.042,Z 511.42,A -85,B 0,C 180,E1 24794.748,E2 24794.748} C_VEL
LIN {X 0,Y 559.388,Z 756.849,A -85,B 0,C 180,E1 24791.203,E2 24791.203} C_VEL
LIN {X 0,Y 556.641,Z 844.126,A -85,B 0,C 180,E1 24789.921,E2 24789.921} C_VEL
LIN {X 0,Y 555.005,Z 869.41,A -85,B 0,C 180,E1 24789.382,E2 24789.382} C_VEL
LIN {X 0,Y 553.136,Z 891.86,A -85,B 0,C 180,E1 24788.741,E2 24788.741} C_VEL
LIN {X 0,Y 550.709,Z 915.905,A -85,B 0,C 180,E1 24787.857,E2 24787.857} C_VEL
LIN {X 0,Y 548.308,Z 936.522,A -85,B 0,C 180,E1 24786.933,E2 24786.933} C_VEL
LIN {X 0,Y 545.245,Z 960.03,A -85,B 0,C 180,E1 24785.669,E2 24785.669} C_VEL
LIN {X 0,Y 542.515,Z 979.131,A -85,B 0,C 180,E1 24784.46,E2 24784.46} C_VEL
LIN {X 0,Y 539.314,Z 1000.359,A -85,B 0,C 180,E1 24782.904,E2 24782.904} C_VEL
LIN {X 0,Y 536.414,Z 1018.716,A -85,B 0,C 180,E1 24781.337,E2 24781.337} C_VEL
LIN {X 0,Y 533.395,Z 1037.817,A -85,B 0,C 180,E1 24779.477,E2 24779.477} C_VEL
LIN {X 0,Y 530.663,Z 1054.689,A -85,B 0,C 180,E1 24777.576,E2 24777.576} C_VEL
LIN {X 0,Y 528.124,Z 1071.281,A -85,B 0,C 180,E1 24775.454,E2 24775.454} C_VEL
LIN {X 0,Y 525.948,Z 1085.828,A -85,B 0,C 180,E1 24773.293,E2 24773.293} C_VEL
LIN {X 0,Y 524.144,Z 1099.334,A -85,B 0,C 180,E1 24771.017,E2 24771.017} C_VEL
LIN {X 0,Y 522.66,Z 1111.377,A -85,B 0,C 180,E1 24768.632,E2 24768.632} C_VEL
LIN {X 0,Y 521.622,Z 1121.31,A -85,B 0,C 180,E1 24766.367,E2 24766.367} C_VEL
LIN {X 0,Y 520.793,Z 1131.034,A -85,B 0,C 180,E1 24763.713,E2 24763.713} C_VEL
LIN {X 0,Y 520.341,Z 1137.816,A -85,B 0,C 180,E1 24761.471,E2 24761.471} C_VEL
LIN {X 0,Y 520.059,Z 1144.198,A -85,B 0,C 180,E1 24758.848,E2 24758.848} C_VEL
LIN {X 0,Y 519.956,Z 1148.522,A -85,B 0,C 180,E1 24756.404,E2 24756.404} C_VEL
LIN {X 0,Y 519.927,Z 1151.396,A -85,B 0,C 180,E1 24754.08,E2 24754.08} C_VEL
LIN {X 0,Y 519.918,Z 1153.132,A -85,B 0,C 180,E1 24751.322,E2 24751.322} C_VEL
LIN {X 0,Y 519.905,Z 1153.226,A -85,B 0,C 180,E1 24749.118,E2 24749.118} C_VEL
LIN {X 0,Y 519.902,Z 1152.219,A -85,B 0,C 180,E1 24746.913,E2 24746.913} C_VEL
LIN {X 0,Y 519.935,Z 1149.514,A -85,B 0,C 180,E1 24744.261,E2 24744.261} C_VEL
LIN {X 0,Y 520.011,Z 1145.694,A -85,B 0,C 180,E1 24741.931,E2 24741.931} C_VEL
LIN {X 0,Y 520.209,Z 1140.608,A -85,B 0,C 180,E1 24739.591,E2 24739.591} C_VEL
LIN {X 0,Y 520.66,Z 1133.031,A -85,B 0,C 180,E1 24736.902,E2 24736.902} C_VEL
LIN {X 0,Y 521.266,Z 1125.243,A -85,B 0,C 180,E1 24734.65,E2 24734.65} C_VEL
LIN {X 0,Y 522.317,Z 1114.564,A -85,B 0,C 180,E1 24732.049,E2 24732.049} C_VEL
LIN {X 0,Y 523.585,Z 1103.497,A -85,B 0,C 180,E1 24729.778,E2 24729.778} C_VEL
LIN {X 0,Y 525.386,Z 1090.038,A -85,B 0,C 180,E1 24727.374,E2 24727.374} C_VEL
LIN {X 0,Y 527.378,Z 1076.017,A -85,B 0,C 180,E1 24725.228,E2 24725.228} C_VEL
LIN {X 0,Y 529.86,Z 1060.048,A -85,B 0,C 180,E1 24723.07,E2 24723.07} C_VEL
LIN {X 0,Y 532.52,Z 1042.93,A -85,B 0,C 180,E1 24721.08,E2 24721.08} C_VEL
LIN {X 0,Y 535.534,Z 1024.472,A -85,B 0,C 180,E1 24719.19,E2 24719.19} C_VEL
LIN {X 0,Y 538.556,Z 1005.079,A -85,B 0,C 180,E1 24717.487,E2 24717.487} C_VEL
LIN {X 0,Y 541.684,Z 984.814,A -85,B 0,C 180,E1 24715.928,E2 24715.928} C_VEL
LIN {X 0,Y 544.72,Z 963.569,A -85,B 0,C 180,E1 24714.546,E2 24714.546} C_VEL
LIN {X 0,Y 547.626,Z 942.048,A -85,B 0,C 180,E1 24713.34,E2 24713.34} C_VEL
LIN {X 0,Y 550.275,Z 919.694,A -85,B 0,C 180,E1 24712.306,E2 24712.306} C_VEL
LIN {X 0,Y 552.404,Z 899.456,A -85,B 0,C 180,E1 24711.522,E2 24711.522} C_VEL
LIN {X 0,Y 554.633,Z 874.335,A -85,B 0,C 180,E1 24710.75,E2 24710.75} C_VEL
LIN {X 0,Y 556.143,Z 852.626,A -85,B 0,C 180,E1 24710.246,E2 24710.246} C_VEL
LIN {X 0,Y 557.433,Z 821.903,A -85,B 0,C 180,E1 24709.738,E2 24709.738} C_VEL
LIN {X 0,Y 564.524,Z 588.106,A -85,B 0,C 180,E1 24706.359,E2 24706.359} C_VEL
LIN {X 0,Y 566.862,Z 510.835,A -85,B 0,C 180,E1 24705.233,E2 24705.233} C_VEL
LIN {X 0,Y 553.338,Z 488.519,A -85,B 0,C 180,E1 24703.51,E2 24703.51} C_VEL
LIN {X 0,Y 540.799,Z 469.555,A -85,B 0,C 180,E1 24701.818,E2 24701.818} C_VEL
LIN {X 0,Y 535.076,Z 461.041,A -85,B 0,C 180,E1 24700.979,E2 24700.979} C_VEL
LIN {X 0,Y 529.274,Z 448.521,A -85,B 0,C 180,E1 24698.845,E2 24698.845} C_VEL
LIN {X 0,Y 525.11,Z 439.956,A -85,B 0,C 180,E1 24697.256,E2 24697.256} C_VEL
LIN {X 0,Y 523.15,Z 435.859,A -85,B 0,C 180,E1 24696.471,E2 24696.471} C_VEL
LIN {X 0,Y 521.749,Z 432.396,A -85,B 0,C 180,E1 24695.768,E2 24695.768} C_VEL
LIN {X 0,Y 521.744,Z 432.188,A -85,B 0,C 180,E1 24692.453,E2 24692.453} C_VEL
LIN {X 0,Y 521.716,Z 432.225,A -85,B 0,C 180,E1 24689.079,E2 24689.079} C_VEL
LIN {X 0,Y 521.715,Z 432.225,A -85,B 0,C 180,E1 24685.545,E2 24685.545} C_VEL
LIN {X 0,Y 521.753,Z 432.217,A -85,B 0,C 180,E1 24682.181,E2 24682.181} C_VEL
LIN {X 0,Y 521.713,Z 432.223,A -85,B 0,C 180,E1 24678.776,E2 24678.776} C_VEL
LIN {X 0,Y 521.703,Z 432.234,A -85,B 0,C 180,E1 24675.337,E2 24675.337} C_VEL
LIN {X 0,Y 521.748,Z 432.242,A -85,B 0,C 180,E1 24671.945,E2 24671.945} C_VEL
LIN {X 0,Y 521.709,Z 432.237,A -85,B 0,C 180,E1 24668.524,E2 24668.524} C_VEL
LIN {X 0,Y 521.688,Z 432.224,A -85,B 0,C 180,E1 24665.058,E2 24665.058} C_VEL
LIN {X 0,Y 521.741,Z 432.221,A -85,B 0,C 180,E1 24661.757,E2 24661.757} C_VEL
LIN {X 0,Y 521.686,Z 432.246,A -85,B 0,C 180,E1 24658.572,E2 24658.572} C_VEL
LIN {X 0,Y 521.685,Z 432.235,A -85,B 0,C 180,E1 24655.052,E2 24655.052} C_VEL
LIN {X 0,Y 521.741,Z 432.216,A -85,B 0,C 180,E1 24651.736,E2 24651.736} C_VEL
LIN {X 0,Y 521.677,Z 432.234,A -85,B 0,C 180,E1 24648.359,E2 24648.359} C_VEL
LIN {X 0,Y 521.675,Z 432.246,A -85,B 0,C 180,E1 24644.89,E2 24644.89} C_VEL
LIN {X 0,Y 521.727,Z 432.238,A -85,B 0,C 180,E1 24641.563,E2 24641.563} C_VEL
LIN {X 0,Y 521.662,Z 432.236,A -85,B 0,C 180,E1 24638.288,E2 24638.288} C_VEL
LIN {X 0,Y 521.679,Z 432.23,A -85,B 0,C 180,E1 24634.939,E2 24634.939} C_VEL
LIN {X 0,Y 521.681,Z 432.229,A -85,B 0,C 180,E1 24631.743,E2 24631.743} C_VEL
LIN {X 0,Y 521.649,Z 432.234,A -85,B 0,C 180,E1 24628.447,E2 24628.447} C_VEL
LIN {X 0,Y 521.7,Z 432.186,A -85,B 0,C 180,E1 24625.116,E2 24625.116} C_VEL
LIN {X 0,Y 521.737,Z 432.419,A -85,B 0,C 180,E1 24623.313,E2 24623.313} C_VEL
LIN {X 0,Y 523.202,Z 436.046,A -85,B 0,C 180,E1 24622.574,E2 24622.574} C_VEL
LIN {X 0,Y 526.259,Z 442.562,A -85,B 0,C 180,E1 24621.31,E2 24621.31} C_VEL
LIN {X 0,Y 531.465,Z 453.843,A -85,B 0,C 180,E1 24619.244,E2 24619.244} C_VEL
LIN {X 0,Y 537.819,Z 468.486,A -85,B 0,C 180,E1 24616.785,E2 24616.785} C_VEL
LIN {X 0,Y 544.881,Z 486.438,A -85,B 0,C 180,E1 24614.066,E2 24614.066} C_VEL
LIN {X 0,Y 547.191,Z 492.131,A -85,B 0,C 180,E1 24613.303,E2 24613.303} C_VEL
LIN {X 0,Y 556.376,Z 507.87,A -85,B 0,C 180,E1 24612.088,E2 24612.088} C_VEL
LIN {X 0,Y 563.927,Z 546.94,A -85,B 0,C 180,E1 24610.707,E2 24610.707} C_VEL
LIN {X 0,Y 557.111,Z 811.193,A -85,B 0,C 180,E1 24607.115,E2 24607.115} C_VEL
LIN {X 0,Y 555.895,Z 851.196,A -85,B 0,C 180,E1 24606.543,E2 24606.543} C_VEL
LIN {X 0,Y 555.344,Z 860.705,A -85,B 0,C 180,E1 24606.354,E2 24606.354} C_VEL
LIN {X 0,Y 553.464,Z 870.469,A -85,B 0,C 180,E1 24606.242,E2 24606.242} C_VEL
LIN {X 0,Y 547.819,Z 887.4,A -85,B 0,C 180,E1 24606.13,E2 24606.13} C_VEL
LIN {X 0,Y 546.337,Z 894.808,A -85,B 0,C 180,E1 24605.954,E2 24605.954} C_VEL
LIN {X 0,Y 544.019,Z 915.942,A -85,B 0,C 180,E1 24605.154,E2 24605.154} C_VEL
LIN {X 0,Y 541.32,Z 937.46,A -85,B 0,C 180,E1 24604.162,E2 24604.162} C_VEL
LIN {X 0,Y 538.36,Z 957.481,A -85,B 0,C 180,E1 24603.033,E2 24603.033} C_VEL
LIN {X 0,Y 535.256,Z 977.163,A -85,B 0,C 180,E1 24601.726,E2 24601.726} C_VEL
LIN {X 0,Y 531.998,Z 995.95,A -85,B 0,C 180,E1 24600.246,E2 24600.246} C_VEL
LIN {X 0,Y 528.522,Z 1015.202,A -85,B 0,C 180,E1 24598.473,E2 24598.473} C_VEL
LIN {X 0,Y 525.513,Z 1031.312,A -85,B 0,C 180,E1 24596.743,E2 24596.743} C_VEL
LIN {X 0,Y 522.411,Z 1047.941,A -85,B 0,C 180,E1 24594.661,E2 24594.661} C_VEL
LIN {X 0,Y 519.822,Z 1062.243,A -85,B 0,C 180,E1 24592.587,E2 24592.587} C_VEL
LIN {X 0,Y 517.528,Z 1075.339,A -85,B 0,C 180,E1 24590.351,E2 24590.351} C_VEL
LIN {X 0,Y 515.716,Z 1086.879,A -85,B 0,C 180,E1 24588.072,E2 24588.072} C_VEL
LIN {X 0,Y 514.274,Z 1096.964,A -85,B 0,C 180,E1 24585.68,E2 24585.68} C_VEL
LIN {X 0,Y 513.23,Z 1105.844,A -85,B 0,C 180,E1 24583.176,E2 24583.176} C_VEL
LIN {X 0,Y 512.586,Z 1112.622,A -85,B 0,C 180,E1 24580.793,E2 24580.793} C_VEL
LIN {X 0,Y 512.181,Z 1118.482,A -85,B 0,C 180,E1 24578.193,E2 24578.193} C_VEL
LIN {X 0,Y 512.003,Z 1122.303,A -85,B 0,C 180,E1 24575.829,E2 24575.829} C_VEL
LIN {X 0,Y 511.94,Z 1125.089,A -85,B 0,C 180,E1 24573.247,E2 24573.247} C_VEL
LIN {X 0,Y 511.927,Z 1126.189,A -85,B 0,C 180,E1 24570.783,E2 24570.783} C_VEL
LIN {X 0,Y 511.925,Z 1125.995,A -85,B 0,C 180,E1 24568.209,E2 24568.209} C_VEL
LIN {X 0,Y 511.956,Z 1124.234,A -85,B 0,C 180,E1 24565.744,E2 24565.744} C_VEL
LIN {X 0,Y 512.056,Z 1121.197,A -85,B 0,C 180,E1 24563.272,E2 24563.272} C_VEL
LIN {X 0,Y 512.307,Z 1116.314,A -85,B 0,C 180,E1 24560.677,E2 24560.677} C_VEL
LIN {X 0,Y 512.801,Z 1110.216,A -85,B 0,C 180,E1 24558.186,E2 24558.186} C_VEL
LIN {X 0,Y 513.615,Z 1102.315,A -85,B 0,C 180,E1 24555.686,E2 24555.686} C_VEL
LIN {X 0,Y 514.857,Z 1092.775,A -85,B 0,C 180,E1 24553.18,E2 24553.18} C_VEL
LIN {X 0,Y 516.407,Z 1082.265,A -85,B 0,C 180,E1 24550.89,E2 24550.89} C_VEL
LIN {X 0,Y 518.541,Z 1069.449,A -85,B 0,C 180,E1 24548.508,E2 24548.508} C_VEL
LIN {X 0,Y 520.836,Z 1056.573,A -85,B 0,C 180,E1 24546.465,E2 24546.465} C_VEL
LIN {X 0,Y 523.755,Z 1040.728,A -85,B 0,C 180,E1 24544.302,E2 24544.302} C_VEL
LIN {X 0,Y 526.801,Z 1024.627,A -85,B 0,C 180,E1 24542.411,E2 24542.411} C_VEL
LIN {X 0,Y 530.047,Z 1006.85,A -85,B 0,C 180,E1 24540.628,E2 24540.628} C_VEL
LIN {X 0,Y 533.387,Z 988.395,A -85,B 0,C 180,E1 24539.03,E2 24539.03} C_VEL
LIN {X 0,Y 536.483,Z 969.684,A -85,B 0,C 180,E1 24537.662,E2 24537.662} C_VEL
LIN {X 0,Y 539.57,Z 949.891,A -85,B 0,C 180,E1 24536.416,E2 24536.416} C_VEL
LIN {X 0,Y 542.4,Z 929.153,A -85,B 0,C 180,E1 24535.34,E2 24535.34} C_VEL
LIN {X 0,Y 545.018,Z 907.508,A -85,B 0,C 180,E1 24534.406,E2 24534.406} C_VEL
LIN {X 0,Y 547.167,Z 885.733,A -85,B 0,C 180,E1 24533.671,E2 24533.671} C_VEL
LIN {X 0,Y 549.017,Z 862.004,A -85,B 0,C 180,E1 24533.061,E2 24533.061} C_VEL
LIN {X 0,Y 550.116,Z 840.4,A -85,B 0,C 180,E1 24532.672,E2 24532.672} C_VEL
LIN {X 0,Y 556.728,Z 592.852,A -85,B 0,C 180,E1 24529.275,E2 24529.275} C_VEL
LIN {X 0,Y 557.917,Z 547.431,A -85,B 0,C 180,E1 24528.632,E2 24528.632} C_VEL
LIN {X 0,Y 550.863,Z 511.532,A -85,B 0,C 180,E1 24527.319,E2 24527.319} C_VEL
LIN {X 0,Y 538.721,Z 491.193,A -85,B 0,C 180,E1 24525.647,E2 24525.647} C_VEL
LIN {X 0,Y 532.51,Z 475.34,A -85,B 0,C 180,E1 24523.264,E2 24523.264} C_VEL
LIN {X 0,Y 526.273,Z 460.781,A -85,B 0,C 180,E1 24520.812,E2 24520.812} C_VEL
LIN {X 0,Y 521.131,Z 449.336,A -85,B 0,C 180,E1 24518.719,E2 24518.719} C_VEL
LIN {X 0,Y 515.367,Z 437.118,A -85,B 0,C 180,E1 24516.281,E2 24516.281} C_VEL
LIN {X 0,Y 513.752,Z 433.425,A -85,B 0,C 180,E1 24515.475,E2 24515.475} C_VEL
LIN {X 0,Y 513.765,Z 433.227,A -85,B 0,C 180,E1 24512.49,E2 24512.49} C_VEL
LIN {X 0,Y 513.724,Z 433.232,A -85,B 0,C 180,E1 24509.245,E2 24509.245} C_VEL
LIN {X 0,Y 513.716,Z 433.235,A -85,B 0,C 180,E1 24505.849,E2 24505.849} C_VEL
LIN {X 0,Y 513.788,Z 433.232,A -85,B 0,C 180,E1 24502.544,E2 24502.544} C_VEL
LIN {X 0,Y 513.726,Z 433.236,A -85,B 0,C 180,E1 24499.204,E2 24499.204} C_VEL
LIN {X 0,Y 513.728,Z 433.227,A -85,B 0,C 180,E1 24495.697,E2 24495.697} C_VEL
LIN {X 0,Y 513.781,Z 433.208,A -85,B 0,C 180,E1 24492.476,E2 24492.476} C_VEL
LIN {X 0,Y 513.73,Z 433.223,A -85,B 0,C 180,E1 24489.184,E2 24489.184} C_VEL
LIN {X 0,Y 513.759,Z 433.233,A -85,B 0,C 180,E1 24485.809,E2 24485.809} C_VEL
LIN {X 0,Y 513.778,Z 433.217,A -85,B 0,C 180,E1 24482.454,E2 24482.454} C_VEL
LIN {X 0,Y 513.739,Z 433.209,A -85,B 0,C 180,E1 24479.219,E2 24479.219} C_VEL
LIN {X 0,Y 513.789,Z 433.22,A -85,B 0,C 180,E1 24475.871,E2 24475.871} C_VEL
LIN {X 0,Y 513.77,Z 433.233,A -85,B 0,C 180,E1 24472.508,E2 24472.508} C_VEL
LIN {X 0,Y 513.754,Z 433.221,A -85,B 0,C 180,E1 24469.118,E2 24469.118} C_VEL
LIN {X 0,Y 513.801,Z 433.205,A -85,B 0,C 180,E1 24465.691,E2 24465.691} C_VEL
LIN {X 0,Y 513.78,Z 433.211,A -85,B 0,C 180,E1 24462.326,E2 24462.326} C_VEL
LIN {X 0,Y 513.764,Z 433.223,A -85,B 0,C 180,E1 24458.897,E2 24458.897} C_VEL
LIN {X 0,Y 513.805,Z 433.225,A -85,B 0,C 180,E1 24455.511,E2 24455.511} C_VEL
LIN {X 0,Y 513.803,Z 433.225,A -85,B 0,C 180,E1 24452.03,E2 24452.03} C_VEL
LIN {X 0,Y 513.776,Z 433.223,A -85,B 0,C 180,E1 24448.69,E2 24448.69} C_VEL
LIN {X 0,Y 513.831,Z 433.391,A -85,B 0,C 180,E1 24445.33,E2 24445.33} C_VEL
LIN {X 0,Y 515.413,Z 437.144,A -85,B 0,C 180,E1 24444.545,E2 24444.545} C_VEL
LIN {X 0,Y 518.733,Z 444.092,A -85,B 0,C 180,E1 24443.168,E2 24443.168} C_VEL
LIN {X 0,Y 522.795,Z 452.525,A -85,B 0,C 180,E1 24441.567,E2 24441.567} C_VEL
LIN {X 0,Y 527.297,Z 461.972,A -85,B 0,C 180,E1 24439.926,E2 24439.926} C_VEL
LIN {X 0,Y 540.391,Z 481.068,A -85,B 0,C 180,E1 24438.019,E2 24438.019} C_VEL
LIN {X 0,Y 554.153,Z 502.668,A -85,B 0,C 180,E1 24436.16,E2 24436.16} C_VEL
LIN {X 0,Y 561.084,Z 514.637,A -85,B 0,C 180,E1 24435.26,E2 24435.26} C_VEL
LIN {X 0,Y 553.163,Z 758.655,A -85,B 0,C 180,E1 24431.704,E2 24431.704} C_VEL
LIN {X 0,Y 550.359,Z 844.119,A -85,B 0,C 180,E1 24430.436,E2 24430.436} C_VEL
LIN {X 0,Y 548.66,Z 869.444,A -85,B 0,C 180,E1 24429.893,E2 24429.893} C_VEL
LIN {X 0,Y 546.714,Z 891.956,A -85,B 0,C 180,E1 24429.245,E2 24429.245} C_VEL
LIN {X 0,Y 544.221,Z 915.713,A -85,B 0,C 180,E1 24428.365,E2 24428.365} C_VEL
LIN {X 0,Y 541.777,Z 935.917,A -85,B 0,C 180,E1 24427.454,E2 24427.454} C_VEL
LIN {X 0,Y 538.592,Z 959.471,A -85,B 0,C 180,E1 24426.183,E2 24426.183} C_VEL
LIN {X 0,Y 535.743,Z 978.662,A -85,B 0,C 180,E1 24424.958,E2 24424.958} C_VEL
LIN {X 0,Y 532.392,Z 999.946,A -85,B 0,C 180,E1 24423.387,E2 24423.387} C_VEL
LIN {X 0,Y 529.295,Z 1018.61,A -85,B 0,C 180,E1 24421.778,E2 24421.778} C_VEL
LIN {X 0,Y 526.216,Z 1037.225,A -85,B 0,C 180,E1 24419.949,E2 24419.949} C_VEL
LIN {X 0,Y 523.282,Z 1054.511,A -85,B 0,C 180,E1 24417.976,E2 24417.976} C_VEL
LIN {X 0,Y 520.625,Z 1070.959,A -85,B 0,C 180,E1 24415.847,E2 24415.847} C_VEL
LIN {X 0,Y 518.271,Z 1085.909,A -85,B 0,C 180,E1 24413.593,E2 24413.593} C_VEL
LIN {X 0,Y 516.333,Z 1099.655,A -85,B 0,C 180,E1 24411.231,E2 24411.231} C_VEL
LIN {X 0,Y 514.772,Z 1111.615,A -85,B 0,C 180,E1 24408.811,E2 24408.811} C_VEL
LIN {X 0,Y 513.605,Z 1122.441,A -85,B 0,C 180,E1 24406.281,E2 24406.281} C_VEL
LIN {X 0,Y 512.809,Z 1131.301,A -85,B 0,C 180,E1 24403.761,E2 24403.761} C_VEL
LIN {X 0,Y 512.343,Z 1138.019,A -85,B 0,C 180,E1 24401.482,E2 24401.482} C_VEL
LIN {X 0,Y 512.054,Z 1144.595,A -85,B 0,C 180,E1 24398.648,E2 24398.648} C_VEL
LIN {X 0,Y 511.956,Z 1148.623,A -85,B 0,C 180,E1 24396.279,E2 24396.279} C_VEL
LIN {X 0,Y 511.922,Z 1151.642,A -85,B 0,C 180,E1 24393.696,E2 24393.696} C_VEL
LIN {X 0,Y 511.918,Z 1152.969,A -85,B 0,C 180,E1 24391.119,E2 24391.119} C_VEL
LIN {X 0,Y 511.913,Z 1152.992,A -85,B 0,C 180,E1 24388.993,E2 24388.993} C_VEL
LIN {X 0,Y 511.919,Z 1151.793,A -85,B 0,C 180,E1 24386.529,E2 24386.529} C_VEL
LIN {X 0,Y 511.958,Z 1148.713,A -85,B 0,C 180,E1 24383.783,E2 24383.783} C_VEL
LIN {X 0,Y 512.052,Z 1144.809,A -85,B 0,C 180,E1 24381.465,E2 24381.465} C_VEL
LIN {X 0,Y 512.315,Z 1138.644,A -85,B 0,C 180,E1 24378.745,E2 24378.745} C_VEL
LIN {X 0,Y 512.783,Z 1131.663,A -85,B 0,C 180,E1 24376.353,E2 24376.353} C_VEL
LIN {X 0,Y 513.564,Z 1122.874,A -85,B 0,C 180,E1 24373.834,E2 24373.834} C_VEL
LIN {X 0,Y 514.714,Z 1112.148,A -85,B 0,C 180,E1 24371.305,E2 24371.305} C_VEL
LIN {X 0,Y 516.153,Z 1100.834,A -85,B 0,C 180,E1 24368.999,E2 24368.999} C_VEL
LIN {X 0,Y 518.113,Z 1086.944,A -85,B 0,C 180,E1 24366.575,E2 24366.575} C_VEL
LIN {X 0,Y 520.225,Z 1073.316,A -85,B 0,C 180,E1 24364.498,E2 24364.498} C_VEL
LIN {X 0,Y 523.042,Z 1055.914,A -85,B 0,C 180,E1 24362.196,E2 24362.196} C_VEL
LIN {X 0,Y 525.711,Z 1040.024,A -85,B 0,C 180,E1 24360.362,E2 24360.362} C_VEL
LIN {X 0,Y 529.011,Z 1020.327,A -85,B 0,C 180,E1 24358.383,E2 24358.383} C_VEL
LIN {X 0,Y 531.92,Z 1002.615,A -85,B 0,C 180,E1 24356.837,E2 24356.837} C_VEL
LIN {X 0,Y 535.482,Z 980.245,A -85,B 0,C 180,E1 24355.153,E2 24355.153} C_VEL
LIN {X 0,Y 538.314,Z 961.229,A -85,B 0,C 180,E1 24353.927,E2 24353.927} C_VEL
LIN {X 0,Y 541.49,Z 938.113,A -85,B 0,C 180,E1 24352.656,E2 24352.656} C_VEL
LIN {X 0,Y 544.102,Z 916.546,A -85,B 0,C 180,E1 24351.674,E2 24351.674} C_VEL
LIN {X 0,Y 546.638,Z 892.562,A -85,B 0,C 180,E1 24350.778,E2 24350.778} C_VEL
LIN {X 0,Y 548.599,Z 869.863,A -85,B 0,C 180,E1 24350.122,E2 24350.122} C_VEL
LIN {X 0,Y 550.299,Z 844.805,A -85,B 0,C 180,E1 24349.579,E2 24349.579} C_VEL
LIN {X 0,Y 552.723,Z 771.886,A -85,B 0,C 180,E1 24348.494,E2 24348.494} C_VEL
LIN {X 0,Y 560.312,Z 535.921,A -85,B 0,C 180,E1 24345.052,E2 24345.052} C_VEL
LIN {X 0,Y 560.908,Z 514.177,A -85,B 0,C 180,E1 24344.724,E2 24344.724} C_VEL
LIN {X 0,Y 547.597,Z 492.181,A -85,B 0,C 180,E1 24342.982,E2 24342.982} C_VEL
LIN {X 0,Y 533.998,Z 471.605,A -85,B 0,C 180,E1 24341.09,E2 24341.09} C_VEL
LIN {X 0,Y 526.995,Z 461.506,A -85,B 0,C 180,E1 24340.031,E2 24340.031} C_VEL
LIN {X 0,Y 521.308,Z 449.323,A -85,B 0,C 180,E1 24337.863,E2 24337.863} C_VEL
LIN {X 0,Y 517.283,Z 441.062,A -85,B 0,C 180,E1 24336.263,E2 24336.263} C_VEL
LIN {X 0,Y 515.35,Z 437.065,A -85,B 0,C 180,E1 24335.459,E2 24335.459} C_VEL
LIN {X 0,Y 513.831,Z 433.381,A -85,B 0,C 180,E1 24334.67,E2 24334.67} C_VEL
LIN {X 0,Y 513.776,Z 433.223,A -85,B 0,C 180,E1 24331.307,E2 24331.307} C_VEL
LIN {X 0,Y 513.797,Z 433.228,A -85,B 0,C 180,E1 24327.844,E2 24327.844} C_VEL
LIN {X 0,Y 513.811,Z 433.225,A -85,B 0,C 180,E1 24324.366,E2 24324.366} C_VEL
LIN {X 0,Y 513.77,Z 433.224,A -85,B 0,C 180,E1 24320.984,E2 24320.984} C_VEL
LIN {X 0,Y 513.769,Z 433.216,A -85,B 0,C 180,E1 24317.44,E2 24317.44} C_VEL
LIN {X 0,Y 513.812,Z 433.203,A -85,B 0,C 180,E1 24314.079,E2 24314.079} C_VEL
LIN {X 0,Y 513.765,Z 433.216,A -85,B 0,C 180,E1 24310.655,E2 24310.655} C_VEL
LIN {X 0,Y 513.756,Z 433.232,A -85,B 0,C 180,E1 24307.155,E2 24307.155} C_VEL
LIN {X 0,Y 513.8,Z 433.223,A -85,B 0,C 180,E1 24303.794,E2 24303.794} C_VEL
LIN {X 0,Y 513.755,Z 433.209,A -85,B 0,C 180,E1 24300.446,E2 24300.446} C_VEL
LIN {X 0,Y 513.743,Z 433.213,A -85,B 0,C 180,E1 24296.988,E2 24296.988} C_VEL
LIN {X 0,Y 513.804,Z 433.226,A -85,B 0,C 180,E1 24293.631,E2 24293.631} C_VEL
LIN {X 0,Y 513.748,Z 433.23,A -85,B 0,C 180,E1 24290.251,E2 24290.251} C_VEL
LIN {X 0,Y 513.733,Z 433.217,A -85,B 0,C 180,E1 24286.837,E2 24286.837} C_VEL
LIN {X 0,Y 513.789,Z 433.21,A -85,B 0,C 180,E1 24283.609,E2 24283.609} C_VEL
LIN {X 0,Y 513.731,Z 433.227,A -85,B 0,C 180,E1 24280.205,E2 24280.205} C_VEL
LIN {X 0,Y 513.727,Z 433.235,A -85,B 0,C 180,E1 24276.727,E2 24276.727} C_VEL
LIN {X 0,Y 513.779,Z 433.234,A -85,B 0,C 180,E1 24273.409,E2 24273.409} C_VEL
LIN {X 0,Y 513.717,Z 433.242,A -85,B 0,C 180,E1 24270.114,E2 24270.114} C_VEL
LIN {X 0,Y 513.716,Z 433.232,A -85,B 0,C 180,E1 24266.576,E2 24266.576} C_VEL
LIN {X 0,Y 513.741,Z 433.429,A -85,B 0,C 180,E1 24264.413,E2 24264.413} C_VEL
LIN {X 0,Y 515.228,Z 436.938,A -85,B 0,C 180,E1 24263.647,E2 24263.647} C_VEL
LIN {X 0,Y 518.449,Z 443.825,A -85,B 0,C 180,E1 24262.255,E2 24262.255} C_VEL
LIN {X 0,Y 521.798,Z 450.712,A -85,B 0,C 180,E1 24260.903,E2 24260.903} C_VEL
LIN {X 0,Y 527.509,Z 463.625,A -85,B 0,C 180,E1 24258.583,E2 24258.583} C_VEL
LIN {X 0,Y 534.182,Z 479.671,A -85,B 0,C 180,E1 24255.954,E2 24255.954} C_VEL
LIN {X 0,Y 538.788,Z 491.403,A -85,B 0,C 180,E1 24254.227,E2 24254.227} C_VEL
LIN {X 0,Y 551.03,Z 511.932,A -85,B 0,C 180,E1 24252.556,E2 24252.556} C_VEL
LIN {X 0,Y 557.992,Z 548.863,A -85,B 0,C 180,E1 24251.237,E2 24251.237} C_VEL
LIN {X 0,Y 550.864,Z 812.559,A -85,B 0,C 180,E1 24247.62,E2 24247.62} C_VEL
LIN {X 0,Y 549.617,Z 851.389,A -85,B 0,C 180,E1 24247.058,E2 24247.058} C_VEL
LIN {X 0,Y 548.115,Z 873.85,A -85,B 0,C 180,E1 24246.565,E2 24246.565} C_VEL
LIN {X 0,Y 546.337,Z 894.808,A -85,B 0,C 180,E1 24245.954,E2 24245.954} C_VEL
LIN {X 0,Y 544.789,Z 902.192,A -85,B 0,C 180,E1 24245.758,E2 24245.758} C_VEL
LIN {X 0,Y 537.804,Z 920.799,A -85,B 0,C 180,E1 24245.403,E2 24245.403} C_VEL
LIN {X 0,Y 536.058,Z 927.892,A -85,B 0,C 180,E1 24245.14,E2 24245.14} C_VEL
LIN {X 0,Y 533.219,Z 947.942,A -85,B 0,C 180,E1 24244.103,E2 24244.103} C_VEL
LIN {X 0,Y 530.006,Z 968.118,A -85,B 0,C 180,E1 24242.846,E2 24242.846} C_VEL
LIN {X 0,Y 526.889,Z 986.264,A -85,B 0,C 180,E1 24241.522,E2 24241.522} C_VEL
LIN {X 0,Y 523.392,Z 1005.108,A -85,B 0,C 180,E1 24239.909,E2 24239.909} C_VEL
LIN {X 0,Y 520.149,Z 1022.088,A -85,B 0,C 180,E1 24238.222,E2 24238.222} C_VEL
LIN {X 0,Y 516.893,Z 1038.663,A -85,B 0,C 180,E1 24236.295,E2 24236.295} C_VEL
LIN {X 0,Y 513.922,Z 1054.021,A -85,B 0,C 180,E1 24234.238,E2 24234.238} C_VEL
LIN {X 0,Y 511.257,Z 1068.017,A -85,B 0,C 180,E1 24232.024,E2 24232.024} C_VEL
LIN {X 0,Y 508.972,Z 1081.028,A -85,B 0,C 180,E1 24229.629,E2 24229.629} C_VEL
LIN {X 0,Y 507.245,Z 1091.644,A -85,B 0,C 180,E1 24227.317,E2 24227.317} C_VEL
LIN {X 0,Y 505.828,Z 1101.857,A -85,B 0,C 180,E1 24224.657,E2 24224.657} C_VEL
LIN {X 0,Y 504.963,Z 1109.504,A -85,B 0,C 180,E1 24222.232,E2 24222.232} C_VEL
LIN {X 0,Y 504.385,Z 1116.098,A -85,B 0,C 180,E1 24219.586,E2 24219.586} C_VEL
LIN {X 0,Y 504.101,Z 1120.698,A -85,B 0,C 180,E1 24217.179,E2 24217.179} C_VEL
LIN {X 0,Y 503.967,Z 1124.14,A -85,B 0,C 180,E1 24214.552,E2 24214.552} C_VEL
LIN {X 0,Y 503.936,Z 1125.955,A -85,B 0,C 180,E1 24212.161,E2 24212.161} C_VEL
LIN {X 0,Y 503.922,Z 1126.461,A -85,B 0,C 180,E1 24209.432,E2 24209.432} C_VEL
LIN {X 0,Y 503.937,Z 1125.55,A -85,B 0,C 180,E1 24207.043,E2 24207.043} C_VEL
LIN {X 0,Y 504.005,Z 1122.953,A -85,B 0,C 180,E1 24204.307,E2 24204.307} C_VEL
LIN {X 0,Y 504.171,Z 1119.263,A -85,B 0,C 180,E1 24201.905,E2 24201.905} C_VEL
LIN {X 0,Y 504.597,Z 1113.383,A -85,B 0,C 180,E1 24199.149,E2 24199.149} C_VEL
LIN {X 0,Y 505.26,Z 1106.7,A -85,B 0,C 180,E1 24196.729,E2 24196.729} C_VEL
LIN {X 0,Y 506.4,Z 1097.559,A -85,B 0,C 180,E1 24194.068,E2 24194.068} C_VEL
LIN {X 0,Y 507.943,Z 1087.319,A -85,B 0,C 180,E1 24191.591,E2 24191.591} C_VEL
LIN {X 0,Y 509.916,Z 1075.477,A -85,B 0,C 180,E1 24189.211,E2 24189.211} C_VEL
LIN {X 0,Y 512.379,Z 1062.13,A -85,B 0,C 180,E1 24186.906,E2 24186.906} C_VEL
LIN {X 0,Y 515.066,Z 1048.058,A -85,B 0,C 180,E1 24184.84,E2 24184.84} C_VEL
LIN {X 0,Y 518.325,Z 1031.412,A -85,B 0,C 180,E1 24182.732,E2 24182.732} C_VEL
LIN {X 0,Y 521.369,Z 1015.836,A -85,B 0,C 180,E1 24181.037,E2 24181.037} C_VEL
LIN {X 0,Y 524.989,Z 996.683,A -85,B 0,C 180,E1 24179.244,E2 24179.244} C_VEL
LIN {X 0,Y 528.285,Z 978.437,A -85,B 0,C 180,E1 24177.784,E2 24177.784} C_VEL
LIN {X 0,Y 531.605,Z 958.407,A -85,B 0,C 180,E1 24176.428,E2 24176.428} C_VEL
LIN {X 0,Y 534.511,Z 939.467,A -85,B 0,C 180,E1 24175.341,E2 24175.341} C_VEL
LIN {X 0,Y 537.389,Z 917.9,A -85,B 0,C 180,E1 24174.316,E2 24174.316} C_VEL
LIN {X 0,Y 539.599,Z 898.648,A -85,B 0,C 180,E1 24173.566,E2 24173.566} C_VEL
LIN {X 0,Y 541.833,Z 874.406,A -85,B 0,C 180,E1 24172.828,E2 24172.828} C_VEL
LIN {X 0,Y 543.367,Z 852.447,A -85,B 0,C 180,E1 24172.338,E2 24172.338} C_VEL
LIN {X 0,Y 544.58,Z 818.343,A -85,B 0,C 180,E1 24171.829,E2 24171.829} C_VEL
LIN {X 0,Y 551.974,Z 556.655,A -85,B 0,C 180,E1 24168.208,E2 24168.208} C_VEL
LIN {X 0,Y 552.013,Z 548.961,A -85,B 0,C 180,E1 24168.08,E2 24168.08} C_VEL
LIN {X 0,Y 545.552,Z 515.7,A -85,B 0,C 180,E1 24166.841,E2 24166.841} C_VEL
LIN {X 0,Y 533.685,Z 495.899,A -85,B 0,C 180,E1 24165.184,E2 24165.184} C_VEL
LIN {X 0,Y 530.191,Z 489.984,A -85,B 0,C 180,E1 24164.628,E2 24164.628} C_VEL
LIN {X 0,Y 523.497,Z 473.328,A -85,B 0,C 180,E1 24161.952,E2 24161.952} C_VEL
LIN {X 0,Y 517.091,Z 458.641,A -85,B 0,C 180,E1 24159.333,E2 24159.333} C_VEL
LIN {X 0,Y 512.936,Z 449.762,A -85,B 0,C 180,E1 24157.6,E2 24157.6} C_VEL
LIN {X 0,Y 509.452,Z 442.322,A -85,B 0,C 180,E1 24156.072,E2 24156.072} C_VEL
LIN {X 0,Y 507.044,Z 437.532,A -85,B 0,C 180,E1 24155.019,E2 24155.019} C_VEL
LIN {X 0,Y 505.824,Z 434.367,A -85,B 0,C 180,E1 24154.281,E2 24154.281} C_VEL
LIN {X 0,Y 505.818,Z 434.208,A -85,B 0,C 180,E1 24150.915,E2 24150.915} C_VEL
LIN {X 0,Y 505.77,Z 434.213,A -85,B 0,C 180,E1 24147.556,E2 24147.556} C_VEL
LIN {X 0,Y 505.8,Z 434.207,A -85,B 0,C 180,E1 24144.155,E2 24144.155} C_VEL
LIN {X 0,Y 505.798,Z 434.204,A -85,B 0,C 180,E1 24140.966,E2 24140.966} C_VEL
LIN {X 0,Y 505.782,Z 434.211,A -85,B 0,C 180,E1 24137.606,E2 24137.606} C_VEL
LIN {X 0,Y 505.838,Z 434.217,A -85,B 0,C 180,E1 24134.188,E2 24134.188} C_VEL
LIN {X 0,Y 505.81,Z 434.221,A -85,B 0,C 180,E1 24130.824,E2 24130.824} C_VEL
LIN {X 0,Y 505.793,Z 434.205,A -85,B 0,C 180,E1 24127.383,E2 24127.383} C_VEL
LIN {X 0,Y 505.848,Z 434.193,A -85,B 0,C 180,E1 24124.081,E2 24124.081} C_VEL
LIN {X 0,Y 505.819,Z 434.216,A -85,B 0,C 180,E1 24120.68,E2 24120.68} C_VEL
LIN {X 0,Y 505.807,Z 434.224,A -85,B 0,C 180,E1 24117.167,E2 24117.167} C_VEL
LIN {X 0,Y 505.846,Z 434.201,A -85,B 0,C 180,E1 24113.759,E2 24113.759} C_VEL
LIN {X 0,Y 505.832,Z 434.198,A -85,B 0,C 180,E1 24110.442,E2 24110.442} C_VEL
LIN {X 0,Y 505.815,Z 434.212,A -85,B 0,C 180,E1 24106.976,E2 24106.976} C_VEL
LIN {X 0,Y 505.858,Z 434.217,A -85,B 0,C 180,E1 24103.581,E2 24103.581} C_VEL
LIN {X 0,Y 505.86,Z 434.214,A -85,B 0,C 180,E1 24100.124,E2 24100.124} C_VEL
LIN {X 0,Y 505.828,Z 434.212,A -85,B 0,C 180,E1 24096.712,E2 24096.712} C_VEL
LIN {X 0,Y 505.85,Z 434.208,A -85,B 0,C 180,E1 24093.213,E2 24093.213} C_VEL
LIN {X 0,Y 505.876,Z 434.207,A -85,B 0,C 180,E1 24089.741,E2 24089.741} C_VEL
LIN {X 0,Y 505.862,Z 434.381,A -85,B 0,C 180,E1 24086.501,E2 24086.501} C_VEL
LIN {X 0,Y 507.42,Z 437.99,A -85,B 0,C 180,E1 24085.696,E2 24085.696} C_VEL
LIN {X 0,Y 508.475,Z 440.181,A -85,B 0,C 180,E1 24085.231,E2 24085.231} C_VEL
LIN {X 0,Y 510.929,Z 445.205,A -85,B 0,C 180,E1 24084.187,E2 24084.187} C_VEL
LIN {X 0,Y 514.895,Z 453.342,A -85,B 0,C 180,E1 24082.567,E2 24082.567} C_VEL
LIN {X 0,Y 519.159,Z 462.366,A -85,B 0,C 180,E1 24080.929,E2 24080.929} C_VEL
LIN {X 0,Y 531.483,Z 480.024,A -85,B 0,C 180,E1 24079.049,E2 24079.049} C_VEL
LIN {X 0,Y 544.095,Z 499.3,A -85,B 0,C 180,E1 24077.267,E2 24077.267} C_VEL
LIN {X 0,Y 555.171,Z 517.872,A -85,B 0,C 180,E1 24075.782,E2 24075.782} C_VEL
LIN {X 0,Y 546.993,Z 760.057,A -85,B 0,C 180,E1 24072.222,E2 24072.222} C_VEL
LIN {X 0,Y 544.12,Z 844.186,A -85,B 0,C 180,E1 24070.962,E2 24070.962} C_VEL
LIN {X 0,Y 542.358,Z 869.541,A -85,B 0,C 180,E1 24070.414,E2 24070.414} C_VEL
LIN {X 0,Y 540.328,Z 892.175,A -85,B 0,C 180,E1 24069.757,E2 24069.757} C_VEL
LIN {X 0,Y 537.715,Z 916.062,A -85,B 0,C 180,E1 24068.862,E2 24068.862} C_VEL
LIN {X 0,Y 535.148,Z 936.467,A -85,B 0,C 180,E1 24067.931,E2 24067.931} C_VEL
LIN {X 0,Y 531.877,Z 959.634,A -85,B 0,C 180,E1 24066.666,E2 24066.666} C_VEL
LIN {X 0,Y 528.938,Z 978.676,A -85,B 0,C 180,E1 24065.437,E2 24065.437} C_VEL
LIN {X 0,Y 525.515,Z 999.544,A -85,B 0,C 180,E1 24063.882,E2 24063.882} C_VEL
LIN {X 0,Y 522.205,Z 1018.558,A -85,B 0,C 180,E1 24062.226,E2 24062.226} C_VEL
LIN {X 0,Y 518.87,Z 1037.759,A -85,B 0,C 180,E1 24060.308,E2 24060.308} C_VEL
LIN {X 0,Y 515.878,Z 1054.649,A -85,B 0,C 180,E1 24058.351,E2 24058.351} C_VEL
LIN {X 0,Y 513.011,Z 1071.436,A -85,B 0,C 180,E1 24056.135,E2 24056.135} C_VEL
LIN {X 0,Y 510.621,Z 1085.928,A -85,B 0,C 180,E1 24053.913,E2 24053.913} C_VEL
LIN {X 0,Y 508.526,Z 1099.959,A -85,B 0,C 180,E1 24051.452,E2 24051.452} C_VEL
LIN {X 0,Y 506.954,Z 1111.336,A -85,B 0,C 180,E1 24049.112,E2 24049.112} C_VEL
LIN {X 0,Y 505.762,Z 1121.699,A -85,B 0,C 180,E1 24046.658,E2 24046.658} C_VEL
LIN {X 0,Y 504.893,Z 1130.68,A -85,B 0,C 180,E1 24044.099,E2 24044.099} C_VEL
LIN {X 0,Y 504.393,Z 1137.458,A -85,B 0,C 180,E1 24041.782,E2 24041.782} C_VEL
LIN {X 0,Y 504.068,Z 1143.933,A -85,B 0,C 180,E1 24039.016,E2 24039.016} C_VEL
LIN {X 0,Y 503.959,Z 1148.232,A -85,B 0,C 180,E1 24036.494,E2 24036.494} C_VEL
LIN {X 0,Y 503.928,Z 1151.195,A -85,B 0,C 180,E1 24033.982,E2 24033.982} C_VEL
LIN {X 0,Y 503.925,Z 1152.735,A -85,B 0,C 180,E1 24031.251,E2 24031.251} C_VEL
LIN {X 0,Y 503.917,Z 1152.782,A -85,B 0,C 180,E1 24028.977,E2 24028.977} C_VEL
LIN {X 0,Y 503.923,Z 1151.579,A -85,B 0,C 180,E1 24026.473,E2 24026.473} C_VEL
LIN {X 0,Y 503.959,Z 1148.56,A -85,B 0,C 180,E1 24023.734,E2 24023.734} C_VEL
LIN {X 0,Y 504.054,Z 1144.575,A -85,B 0,C 180,E1 24021.329,E2 24021.329} C_VEL
LIN {X 0,Y 504.338,Z 1138.395,A -85,B 0,C 180,E1 24018.565,E2 24018.565} C_VEL
LIN {X 0,Y 504.836,Z 1131.406,A -85,B 0,C 180,E1 24016.134,E2 24016.134} C_VEL
LIN {X 0,Y 505.688,Z 1122.462,A -85,B 0,C 180,E1 24013.534,E2 24013.534} C_VEL
LIN {X 0,Y 506.891,Z 1111.867,A -85,B 0,C 180,E1 24011.005,E2 24011.005} C_VEL
LIN {X 0,Y 508.433,Z 1100.546,A -85,B 0,C 180,E1 24008.665,E2 24008.665} C_VEL
LIN {X 0,Y 510.505,Z 1086.636,A -85,B 0,C 180,E1 24006.204,E2 24006.204} C_VEL
LIN {X 0,Y 512.731,Z 1072.999,A -85,B 0,C 180,E1 24004.098,E2 24004.098} C_VEL
LIN {X 0,Y 515.708,Z 1055.572,A -85,B 0,C 180,E1 24001.765,E2 24001.765} C_VEL
LIN {X 0,Y 518.51,Z 1039.67,A -85,B 0,C 180,E1 23999.908,E2 23999.908} C_VEL
LIN {X 0,Y 521.991,Z 1019.753,A -85,B 0,C 180,E1 23997.889,E2 23997.889} C_VEL
LIN {X 0,Y 525.136,Z 1001.525,A -85,B 0,C 180,E1 23996.287,E2 23996.287} C_VEL
LIN {X 0,Y 528.741,Z 979.777,A -85,B 0,C 180,E1 23994.643,E2 23994.643} C_VEL
LIN {X 0,Y 531.689,Z 960.726,A -85,B 0,C 180,E1 23993.405,E2 23993.405} C_VEL
LIN {X 0,Y 534.994,Z 937.507,A -85,B 0,C 180,E1 23992.123,E2 23992.123} C_VEL
LIN {X 0,Y 537.573,Z 917.038,A -85,B 0,C 180,E1 23991.184,E2 23991.184} C_VEL
LIN {X 0,Y 540.191,Z 893.415,A -85,B 0,C 180,E1 23990.287,E2 23990.287} C_VEL
LIN {X 0,Y 542.267,Z 870.262,A -85,B 0,C 180,E1 23989.609,E2 23989.609} C_VEL
LIN {X 0,Y 544.03,Z 845.457,A -85,B 0,C 180,E1 23989.063,E2 23989.063} C_VEL
LIN {X 0,Y 546.277,Z 781.192,A -85,B 0,C 180,E1 23988.093,E2 23988.093} C_VEL
LIN {X 0,Y 554.02,Z 549.165,A -85,B 0,C 180,E1 23984.678,E2 23984.678} C_VEL
LIN {X 0,Y 555.003,Z 517.478,A -85,B 0,C 180,E1 23984.204,E2 23984.204} C_VEL
LIN {X 0,Y 542.276,Z 496.538,A -85,B 0,C 180,E1 23982.497,E2 23982.497} C_VEL
LIN {X 0,Y 529.71,Z 477.4,A -85,B 0,C 180,E1 23980.706,E2 23980.706} C_VEL
LIN {X 0,Y 518.972,Z 462.069,A -85,B 0,C 180,E1 23979.052,E2 23979.052} C_VEL
LIN {X 0,Y 513.698,Z 450.871,A -85,B 0,C 180,E1 23976.974,E2 23976.974} C_VEL
LIN {X 0,Y 509.505,Z 442.291,A -85,B 0,C 180,E1 23975.238,E2 23975.238} C_VEL
LIN {X 0,Y 507.354,Z 437.901,A -85,B 0,C 180,E1 23974.309,E2 23974.309} C_VEL
LIN {X 0,Y 505.863,Z 434.379,A -85,B 0,C 180,E1 23973.499,E2 23973.499} C_VEL
LIN {X 0,Y 505.877,Z 434.205,A -85,B 0,C 180,E1 23970.135,E2 23970.135} C_VEL
LIN {X 0,Y 505.86,Z 434.205,A -85,B 0,C 180,E1 23966.66,E2 23966.66} C_VEL
LIN {X 0,Y 505.829,Z 434.209,A -85,B 0,C 180,E1 23963.165,E2 23963.165} C_VEL
LIN {X 0,Y 505.853,Z 434.213,A -85,B 0,C 180,E1 23959.756,E2 23959.756} C_VEL
LIN {X 0,Y 505.867,Z 434.216,A -85,B 0,C 180,E1 23956.301,E2 23956.301} C_VEL
LIN {X 0,Y 505.82,Z 434.213,A -85,B 0,C 180,E1 23952.907,E2 23952.907} C_VEL
LIN {X 0,Y 505.829,Z 434.199,A -85,B 0,C 180,E1 23949.443,E2 23949.443} C_VEL
LIN {X 0,Y 505.86,Z 434.198,A -85,B 0,C 180,E1 23946.127,E2 23946.127} C_VEL
LIN {X 0,Y 505.812,Z 434.223,A -85,B 0,C 180,E1 23942.719,E2 23942.719} C_VEL
LIN {X 0,Y 505.817,Z 434.218,A -85,B 0,C 180,E1 23939.207,E2 23939.207} C_VEL
LIN {X 0,Y 505.855,Z 434.193,A -85,B 0,C 180,E1 23935.806,E2 23935.806} C_VEL
LIN {X 0,Y 505.8,Z 434.204,A -85,B 0,C 180,E1 23932.503,E2 23932.503} C_VEL
LIN {X 0,Y 505.803,Z 434.22,A -85,B 0,C 180,E1 23928.945,E2 23928.945} C_VEL
LIN {X 0,Y 505.866,Z 434.217,A -85,B 0,C 180,E1 23925.579,E2 23925.579} C_VEL
LIN {X 0,Y 505.798,Z 434.212,A -85,B 0,C 180,E1 23922.157,E2 23922.157} C_VEL
LIN {X 0,Y 505.784,Z 434.207,A -85,B 0,C 180,E1 23918.669,E2 23918.669} C_VEL
LIN {X 0,Y 505.839,Z 434.2,A -85,B 0,C 180,E1 23915.349,E2 23915.349} C_VEL
LIN {X 0,Y 505.789,Z 434.208,A -85,B 0,C 180,E1 23911.933,E2 23911.933} C_VEL
LIN {X 0,Y 505.772,Z 434.211,A -85,B 0,C 180,E1 23908.438,E2 23908.438} C_VEL
LIN {X 0,Y 505.842,Z 434.451,A -85,B 0,C 180,E1 23905.543,E2 23905.543} C_VEL
LIN {X 0,Y 507.663,Z 438.465,A -85,B 0,C 180,E1 23904.629,E2 23904.629} C_VEL
LIN {X 0,Y 510.553,Z 444.656,A -85,B 0,C 180,E1 23903.321,E2 23903.321} C_VEL
LIN {X 0,Y 515.831,Z 455.755,A -85,B 0,C 180,E1 23901.094,E2 23901.094} C_VEL
LIN {X 0,Y 522.42,Z 470.704,A -85,B 0,C 180,E1 23898.383,E2 23898.383} C_VEL
LIN {X 0,Y 529.493,Z 488.298,A -85,B 0,C 180,E1 23895.525,E2 23895.525} C_VEL
LIN {X 0,Y 530.932,Z 491.511,A -85,B 0,C 180,E1 23895.109,E2 23895.109} C_VEL
LIN {X 0,Y 542.041,Z 509.804,A -85,B 0,C 180,E1 23893.534,E2 23893.534} C_VEL
LIN {X 0,Y 545.847,Z 516.631,A -85,B 0,C 180,E1 23893.009,E2 23893.009} C_VEL
LIN {X 0,Y 552.112,Z 550.57,A -85,B 0,C 180,E1 23891.782,E2 23891.782} C_VEL
LIN {X 0,Y 544.668,Z 813.644,A -85,B 0,C 180,E1 23888.141,E2 23888.141} C_VEL
LIN {X 0,Y 543.386,Z 851.567,A -85,B 0,C 180,E1 23887.585,E2 23887.585} C_VEL
LIN {X 0,Y 541.829,Z 873.995,A -85,B 0,C 180,E1 23887.088,E2 23887.088} C_VEL
LIN {X 0,Y 539.729,Z 897.207,A -85,B 0,C 180,E1 23886.391,E2 23886.391} C_VEL
LIN {X 0,Y 537.432,Z 917.286,A -85,B 0,C 180,E1 23885.615,E2 23885.615} C_VEL
LIN {X 0,Y 536.058,Z 927.892,A -85,B 0,C 180,E1 23885.14,E2 23885.14} C_VEL
LIN {X 0,Y 534.271,Z 935.207,A -85,B 0,C 180,E1 23884.855,E2 23884.855} C_VEL
LIN {X 0,Y 526.7,Z 952.954,A -85,B 0,C 180,E1 23884.264,E2 23884.264} C_VEL
LIN {X 0,Y 524.786,Z 959.576,A -85,B 0,C 180,E1 23883.918,E2 23883.918} C_VEL
LIN {X 0,Y 521.064,Z 980.886,A -85,B 0,C 180,E1 23882.435,E2 23882.435} C_VEL
LIN {X 0,Y 517.683,Z 998.963,A -85,B 0,C 180,E1 23880.954,E2 23880.954} C_VEL
LIN {X 0,Y 514.1,Z 1016.987,A -85,B 0,C 180,E1 23879.221,E2 23879.221} C_VEL
LIN {X 0,Y 510.758,Z 1033.468,A -85,B 0,C 180,E1 23877.391,E2 23877.391} C_VEL
LIN {X 0,Y 507.647,Z 1048.552,A -85,B 0,C 180,E1 23875.429,E2 23875.429} C_VEL
LIN {X 0,Y 504.845,Z 1062.593,A -85,B 0,C 180,E1 23873.336,E2 23873.336} C_VEL
LIN {X 0,Y 502.262,Z 1075.89,A -85,B 0,C 180,E1 23870.998,E2 23870.998} C_VEL
LIN {X 0,Y 500.146,Z 1087.901,A -85,B 0,C 180,E1 23868.534,E2 23868.534} C_VEL
LIN {X 0,Y 498.594,Z 1097.652,A -85,B 0,C 180,E1 23866.137,E2 23866.137} C_VEL
LIN {X 0,Y 497.397,Z 1106.664,A -85,B 0,C 180,E1 23863.485,E2 23863.485} C_VEL
LIN {X 0,Y 496.681,Z 1113.38,A -85,B 0,C 180,E1 23861.026,E2 23861.026} C_VEL
LIN {X 0,Y 496.206,Z 1119.325,A -85,B 0,C 180,E1 23858.226,E2 23858.226} C_VEL
LIN {X 0,Y 496.015,Z 1123.045,A -85,B 0,C 180,E1 23855.785,E2 23855.785} C_VEL
LIN {X 0,Y 495.945,Z 1125.708,A -85,B 0,C 180,E1 23853.005,E2 23853.005} C_VEL
LIN {X 0,Y 495.93,Z 1126.653,A -85,B 0,C 180,E1 23850.578,E2 23850.578} C_VEL
LIN {X 0,Y 495.937,Z 1126.219,A -85,B 0,C 180,E1 23847.805,E2 23847.805} C_VEL
LIN {X 0,Y 495.967,Z 1124.442,A -85,B 0,C 180,E1 23845.375,E2 23845.375} C_VEL
LIN {X 0,Y 496.114,Z 1121.078,A -85,B 0,C 180,E1 23842.705,E2 23842.705} C_VEL
LIN {X 0,Y 496.41,Z 1116.518,A -85,B 0,C 180,E1 23840.259,E2 23840.259} C_VEL
LIN {X 0,Y 497.019,Z 1110.012,A -85,B 0,C 180,E1 23837.569,E2 23837.569} C_VEL
LIN {X 0,Y 497.925,Z 1102.407,A -85,B 0,C 180,E1 23835.106,E2 23835.106} C_VEL
LIN {X 0,Y 499.342,Z 1092.786,A -85,B 0,C 180,E1 23832.521,E2 23832.521} C_VEL
LIN {X 0,Y 501.116,Z 1082.277,A -85,B 0,C 180,E1 23830.171,E2 23830.171} C_VEL
LIN {X 0,Y 503.644,Z 1068.642,A -85,B 0,C 180,E1 23827.593,E2 23827.593} C_VEL
LIN {X 0,Y 506.228,Z 1055.645,A -85,B 0,C 180,E1 23825.494,E2 23825.494} C_VEL
LIN {X 0,Y 509.301,Z 1040.571,A -85,B 0,C 180,E1 23823.409,E2 23823.409} C_VEL
LIN {X 0,Y 512.45,Z 1025.275,A -85,B 0,C 180,E1 23821.569,E2 23821.569} C_VEL
LIN {X 0,Y 515.992,Z 1007.566,A -85,B 0,C 180,E1 23819.746,E2 23819.746} C_VEL
LIN {X 0,Y 519.607,Z 989.172,A -85,B 0,C 180,E1 23818.114,E2 23818.114} C_VEL
LIN {X 0,Y 523.132,Z 969.475,A -85,B 0,C 180,E1 23816.644,E2 23816.644} C_VEL
LIN {X 0,Y 526.418,Z 949.93,A -85,B 0,C 180,E1 23815.394,E2 23815.394} C_VEL
LIN {X 0,Y 529.498,Z 929.002,A -85,B 0,C 180,E1 23814.292,E2 23814.292} C_VEL
LIN {X 0,Y 532.38,Z 906.755,A -85,B 0,C 180,E1 23813.326,E2 23813.326} C_VEL
LIN {X 0,Y 534.625,Z 885.552,A -85,B 0,C 180,E1 23812.604,E2 23812.604} C_VEL
LIN {X 0,Y 536.609,Z 861.642,A -85,B 0,C 180,E1 23811.983,E2 23811.983} C_VEL
LIN {X 0,Y 537.783,Z 839.998,A -85,B 0,C 180,E1 23811.589,E2 23811.589} C_VEL
LIN {X 0,Y 545.062,Z 591.54,A -85,B 0,C 180,E1 23808.116,E2 23808.116} C_VEL
LIN {X 0,Y 546.218,Z 550.789,A -85,B 0,C 180,E1 23807.527,E2 23807.527} C_VEL
LIN {X 0,Y 540.356,Z 520.005,A -85,B 0,C 180,E1 23806.365,E2 23806.365} C_VEL
LIN {X 0,Y 529.055,Z 501.128,A -85,B 0,C 180,E1 23804.75,E2 23804.75} C_VEL
LIN {X 0,Y 521.858,Z 489.382,A -85,B 0,C 180,E1 23803.612,E2 23803.612} C_VEL
LIN {X 0,Y 514.907,Z 472.254,A -85,B 0,C 180,E1 23800.729,E2 23800.729} C_VEL
LIN {X 0,Y 508.229,Z 457.044,A -85,B 0,C 180,E1 23797.867,E2 23797.867} C_VEL
LIN {X 0,Y 503.562,Z 447.505,A -85,B 0,C 180,E1 23795.857,E2 23795.857} C_VEL
LIN {X 0,Y 501.196,Z 442.703,A -85,B 0,C 180,E1 23794.79,E2 23794.79} C_VEL
LIN {X 0,Y 499.424,Z 439.056,A -85,B 0,C 180,E1 23793.958,E2 23793.958} C_VEL
LIN {X 0,Y 497.898,Z 435.42,A -85,B 0,C 180,E1 23793.093,E2 23793.093} C_VEL
LIN {X 0,Y 497.836,Z 435.221,A -85,B 0,C 180,E1 23789.742,E2 23789.742} C_VEL
LIN {X 0,Y 497.877,Z 435.215,A -85,B 0,C 180,E1 23786.349,E2 23786.349} C_VEL
LIN {X 0,Y 497.865,Z 435.214,A -85,B 0,C 180,E1 23782.931,E2 23782.931} C_VEL
LIN {X 0,Y 497.842,Z 435.21,A -85,B 0,C 180,E1 23779.476,E2 23779.476} C_VEL
LIN {X 0,Y 497.877,Z 435.193,A -85,B 0,C 180,E1 23776.09,E2 23776.09} C_VEL
LIN {X 0,Y 497.864,Z 435.19,A -85,B 0,C 180,E1 23772.881,E2 23772.881} C_VEL
LIN {X 0,Y 497.853,Z 435.205,A -85,B 0,C 180,E1 23769.479,E2 23769.479} C_VEL
LIN {X 0,Y 497.913,Z 435.209,A -85,B 0,C 180,E1 23766.11,E2 23766.11} C_VEL
LIN {X 0,Y 497.881,Z 435.193,A -85,B 0,C 180,E1 23762.648,E2 23762.648} C_VEL
LIN {X 0,Y 497.861,Z 435.185,A -85,B 0,C 180,E1 23759.194,E2 23759.194} C_VEL
LIN {X 0,Y 497.899,Z 435.196,A -85,B 0,C 180,E1 23755.739,E2 23755.739} C_VEL
LIN {X 0,Y 497.916,Z 435.211,A -85,B 0,C 180,E1 23752.268,E2 23752.268} C_VEL
LIN {X 0,Y 497.879,Z 435.204,A -85,B 0,C 180,E1 23748.767,E2 23748.767} C_VEL
LIN {X 0,Y 497.887,Z 435.188,A -85,B 0,C 180,E1 23745.223,E2 23745.223} C_VEL
LIN {X 0,Y 497.929,Z 435.18,A -85,B 0,C 180,E1 23741.775,E2 23741.775} C_VEL
LIN {X 0,Y 497.905,Z 435.188,A -85,B 0,C 180,E1 23738.315,E2 23738.315} C_VEL
LIN {X 0,Y 497.89,Z 435.193,A -85,B 0,C 180,E1 23734.802,E2 23734.802} C_VEL
LIN {X 0,Y 497.926,Z 435.19,A -85,B 0,C 180,E1 23731.318,E2 23731.318} C_VEL
LIN {X 0,Y 497.956,Z 435.366,A -85,B 0,C 180,E1 23727.743,E2 23727.743} C_VEL
LIN {X 0,Y 499.511,Z 439.058,A -85,B 0,C 180,E1 23726.874,E2 23726.874} C_VEL
LIN {X 0,Y 502.797,Z 445.574,A -85,B 0,C 180,E1 23725.417,E2 23725.417} C_VEL
LIN {X 0,Y 507.307,Z 454.967,A -85,B 0,C 180,E1 23723.47,E2 23723.47} C_VEL
LIN {X 0,Y 511.098,Z 462.809,A -85,B 0,C 180,E1 23721.975,E2 23721.975} C_VEL
LIN {X 0,Y 523.757,Z 480.687,A -85,B 0,C 180,E1 23719.957,E2 23719.957} C_VEL
LIN {X 0,Y 536.613,Z 500.15,A -85,B 0,C 180,E1 23718.068,E2 23718.068} C_VEL
LIN {X 0,Y 548.96,Z 520.466,A -85,B 0,C 180,E1 23716.362,E2 23716.362} C_VEL
LIN {X 0,Y 549.285,Z 521.683,A -85,B 0,C 180,E1 23716.307,E2 23716.307} C_VEL
LIN {X 0,Y 540.85,Z 762.08,A -85,B 0,C 180,E1 23712.743,E2 23712.743} C_VEL
LIN {X 0,Y 537.925,Z 844.361,A -85,B 0,C 180,E1 23711.499,E2 23711.499} C_VEL
LIN {X 0,Y 536.106,Z 869.621,A -85,B 0,C 180,E1 23710.948,E2 23710.948} C_VEL
LIN {X 0,Y 533.997,Z 892.298,A -85,B 0,C 180,E1 23710.285,E2 23710.285} C_VEL
LIN {X 0,Y 531.24,Z 916.515,A -85,B 0,C 180,E1 23709.368,E2 23709.368} C_VEL
LIN {X 0,Y 528.413,Z 938.167,A -85,B 0,C 180,E1 23708.365,E2 23708.365} C_VEL
LIN {X 0,Y 525.017,Z 960.98,A -85,B 0,C 180,E1 23707.088,E2 23707.088} C_VEL
LIN {X 0,Y 521.921,Z 980.224,A -85,B 0,C 180,E1 23705.823,E2 23705.823} C_VEL
LIN {X 0,Y 518.036,Z 1002.58,A -85,B 0,C 180,E1 23704.102,E2 23704.102} C_VEL
LIN {X 0,Y 514.775,Z 1020.663,A -85,B 0,C 180,E1 23702.485,E2 23702.485} C_VEL
LIN {X 0,Y 511.149,Z 1040.395,A -85,B 0,C 180,E1 23700.441,E2 23700.441} C_VEL
LIN {X 0,Y 508.235,Z 1056.215,A -85,B 0,C 180,E1 23698.56,E2 23698.56} C_VEL
LIN {X 0,Y 505.125,Z 1073.502,A -85,B 0,C 180,E1 23696.195,E2 23696.195} C_VEL
LIN {X 0,Y 502.803,Z 1087.07,A -85,B 0,C 180,E1 23694.059,E2 23694.059} C_VEL
LIN {X 0,Y 500.518,Z 1101.57,A -85,B 0,C 180,E1 23691.419,E2 23691.419} C_VEL
LIN {X 0,Y 499.016,Z 1112.126,A -85,B 0,C 180,E1 23689.185,E2 23689.185} C_VEL
LIN {X 0,Y 497.739,Z 1122.773,A -85,B 0,C 180,E1 23686.574,E2 23686.574} C_VEL
LIN {X 0,Y 496.896,Z 1131.174,A -85,B 0,C 180,E1 23684.088,E2 23684.088} C_VEL
LIN {X 0,Y 496.367,Z 1138.156,A -85,B 0,C 180,E1 23681.621,E2 23681.621} C_VEL
LIN {X 0,Y 496.058,Z 1144.347,A -85,B 0,C 180,E1 23678.812,E2 23678.812} C_VEL
LIN {X 0,Y 495.959,Z 1148.177,A -85,B 0,C 180,E1 23676.483,E2 23676.483} C_VEL
LIN {X 0,Y 495.927,Z 1151.212,A -85,B 0,C 180,E1 23673.815,E2 23673.815} C_VEL
LIN {X 0,Y 495.925,Z 1152.549,A -85,B 0,C 180,E1 23671.155,E2 23671.155} C_VEL
LIN {X 0,Y 495.92,Z 1152.572,A -85,B 0,C 180,E1 23668.96,E2 23668.96} C_VEL
LIN {X 0,Y 495.924,Z 1151.359,A -85,B 0,C 180,E1 23666.405,E2 23666.405} C_VEL
LIN {X 0,Y 495.959,Z 1148.34,A -85,B 0,C 180,E1 23663.634,E2 23663.634} C_VEL
LIN {X 0,Y 496.055,Z 1144.561,A -85,B 0,C 180,E1 23661.305,E2 23661.305} C_VEL
LIN {X 0,Y 496.334,Z 1138.78,A -85,B 0,C 180,E1 23658.613,E2 23658.613} C_VEL
LIN {X 0,Y 496.866,Z 1131.521,A -85,B 0,C 180,E1 23656.026,E2 23656.026} C_VEL
LIN {X 0,Y 497.692,Z 1123.187,A -85,B 0,C 180,E1 23653.544,E2 23653.544} C_VEL
LIN {X 0,Y 498.951,Z 1112.653,A -85,B 0,C 180,E1 23650.934,E2 23650.934} C_VEL
LIN {X 0,Y 500.443,Z 1102.035,A -85,B 0,C 180,E1 23648.676,E2 23648.676} C_VEL
LIN {X 0,Y 502.683,Z 1087.775,A -85,B 0,C 180,E1 23646.06,E2 23646.06} C_VEL
LIN {X 0,Y 504.98,Z 1074.271,A -85,B 0,C 180,E1 23643.923,E2 23643.923} C_VEL
LIN {X 0,Y 508.061,Z 1057.133,A -85,B 0,C 180,E1 23641.558,E2 23641.558} C_VEL
LIN {X 0,Y 510.998,Z 1041.139,A -85,B 0,C 180,E1 23639.647,E2 23639.647} C_VEL
LIN {X 0,Y 514.452,Z 1022.474,A -85,B 0,C 180,E1 23637.69,E2 23637.69} C_VEL
LIN {X 0,Y 517.784,Z 1003.842,A -85,B 0,C 180,E1 23636.01,E2 23636.01} C_VEL
LIN {X 0,Y 521.378,Z 983.425,A -85,B 0,C 180,E1 23634.404,E2 23634.404} C_VEL
LIN {X 0,Y 524.682,Z 962.969,A -85,B 0,C 180,E1 23633.04,E2 23633.04} C_VEL
LIN {X 0,Y 527.798,Z 942.441,A -85,B 0,C 180,E1 23631.859,E2 23631.859} C_VEL
LIN {X 0,Y 530.758,Z 920.26,A -85,B 0,C 180,E1 23630.799,E2 23630.799} C_VEL
LIN {X 0,Y 533.138,Z 900.14,A -85,B 0,C 180,E1 23629.997,E2 23629.997} C_VEL
LIN {X 0,Y 535.616,Z 875.315,A -85,B 0,C 180,E1 23629.208,E2 23629.208} C_VEL
LIN {X 0,Y 537.338,Z 853.066,A -85,B 0,C 180,E1 23628.677,E2 23628.677} C_VEL
LIN {X 0,Y 538.735,Z 824.06,A -85,B 0,C 180,E1 23628.18,E2 23628.18} C_VEL
LIN {X 0,Y 546.735,Z 590.547,A -85,B 0,C 180,E1 23624.714,E2 23624.714} C_VEL
LIN {X 0,Y 549.16,Z 520.856,A -85,B 0,C 180,E1 23623.677,E2 23623.677} C_VEL
LIN {X 0,Y 536.028,Z 499.214,A -85,B 0,C 180,E1 23621.862,E2 23621.862} C_VEL
LIN {X 0,Y 522.515,Z 478.888,A -85,B 0,C 180,E1 23619.871,E2 23619.871} C_VEL
LIN {X 0,Y 510.887,Z 462.421,A -85,B 0,C 180,E1 23617.991,E2 23617.991} C_VEL
LIN {X 0,Y 505.567,Z 451.329,A -85,B 0,C 180,E1 23615.817,E2 23615.817} C_VEL
LIN {X 0,Y 501.845,Z 443.6,A -85,B 0,C 180,E1 23614.185,E2 23614.185} C_VEL
LIN {X 0,Y 499.439,Z 438.964,A -85,B 0,C 180,E1 23613.131,E2 23613.131} C_VEL
LIN {X 0,Y 497.955,Z 435.354,A -85,B 0,C 180,E1 23612.285,E2 23612.285} C_VEL
LIN {X 0,Y 497.915,Z 435.19,A -85,B 0,C 180,E1 23608.813,E2 23608.813} C_VEL
LIN {X 0,Y 497.892,Z 435.192,A -85,B 0,C 180,E1 23605.325,E2 23605.325} C_VEL
LIN {X 0,Y 497.915,Z 435.185,A -85,B 0,C 180,E1 23601.809,E2 23601.809} C_VEL
LIN {X 0,Y 497.924,Z 435.181,A -85,B 0,C 180,E1 23598.378,E2 23598.378} C_VEL
LIN {X 0,Y 497.882,Z 435.192,A -85,B 0,C 180,E1 23594.985,E2 23594.985} C_VEL
LIN {X 0,Y 497.894,Z 435.206,A -85,B 0,C 180,E1 23591.468,E2 23591.468} C_VEL
LIN {X 0,Y 497.937,Z 435.204,A -85,B 0,C 180,E1 23587.964,E2 23587.964} C_VEL
LIN {X 0,Y 497.884,Z 435.193,A -85,B 0,C 180,E1 23584.492,E2 23584.492} C_VEL
LIN {X 0,Y 497.869,Z 435.185,A -85,B 0,C 180,E1 23581.036,E2 23581.036} C_VEL
LIN {X 0,Y 497.917,Z 435.196,A -85,B 0,C 180,E1 23577.698,E2 23577.698} C_VEL
LIN {X 0,Y 497.881,Z 435.21,A -85,B 0,C 180,E1 23574.237,E2 23574.237} C_VEL
LIN {X 0,Y 497.857,Z 435.198,A -85,B 0,C 180,E1 23570.754,E2 23570.754} C_VEL
LIN {X 0,Y 497.895,Z 435.185,A -85,B 0,C 180,E1 23567.356,E2 23567.356} C_VEL
LIN {X 0,Y 497.864,Z 435.199,A -85,B 0,C 180,E1 23564.149,E2 23564.149} C_VEL
LIN {X 0,Y 497.85,Z 435.213,A -85,B 0,C 180,E1 23560.647,E2 23560.647} C_VEL
LIN {X 0,Y 497.889,Z 435.213,A -85,B 0,C 180,E1 23557.195,E2 23557.195} C_VEL
LIN {X 0,Y 497.869,Z 435.213,A -85,B 0,C 180,E1 23553.779,E2 23553.779} C_VEL
LIN {X 0,Y 497.837,Z 435.216,A -85,B 0,C 180,E1 23550.39,E2 23550.39} C_VEL
LIN {X 0,Y 497.88,Z 435.243,A -85,B 0,C 180,E1 23547.026,E2 23547.026} C_VEL
LIN {X 0,Y 497.939,Z 435.784,A -85,B 0,C 180,E1 23546.686,E2 23546.686} C_VEL
LIN {X 0,Y 499.456,Z 439.103,A -85,B 0,C 180,E1 23545.906,E2 23545.906} C_VEL
LIN {X 0,Y 502.585,Z 445.508,A -85,B 0,C 180,E1 23544.46,E2 23544.46} C_VEL
LIN {X 0,Y 506.319,Z 453.141,A -85,B 0,C 180,E1 23542.822,E2 23542.822} C_VEL
LIN {X 0,Y 512.992,Z 467.782,A -85,B 0,C 180,E1 23539.968,E2 23539.968} C_VEL
LIN {X 0,Y 520.184,Z 485.089,A -85,B 0,C 180,E1 23536.97,E2 23536.97} C_VEL
LIN {X 0,Y 522.478,Z 490.704,A -85,B 0,C 180,E1 23536.13,E2 23536.13} C_VEL
LIN {X 0,Y 534.819,Z 510.69,A -85,B 0,C 180,E1 23534.309,E2 23534.309} C_VEL
LIN {X 0,Y 540.615,Z 520.901,A -85,B 0,C 180,E1 23533.488,E2 23533.488} C_VEL
LIN {X 0,Y 546.28,Z 552.359,A -85,B 0,C 180,E1 23532.338,E2 23532.338} C_VEL
LIN {X 0,Y 538.525,Z 814.45,A -85,B 0,C 180,E1 23528.677,E2 23528.677} C_VEL
LIN {X 0,Y 537.213,Z 851.567,A -85,B 0,C 180,E1 23528.128,E2 23528.128} C_VEL
LIN {X 0,Y 535.599,Z 873.948,A -85,B 0,C 180,E1 23527.629,E2 23527.629} C_VEL
LIN {X 0,Y 533.421,Z 897.216,A -85,B 0,C 180,E1 23526.926,E2 23526.926} C_VEL
LIN {X 0,Y 531.074,Z 917.018,A -85,B 0,C 180,E1 23526.156,E2 23526.156} C_VEL
LIN {X 0,Y 528.09,Z 938.851,A -85,B 0,C 180,E1 23525.119,E2 23525.119} C_VEL
LIN {X 0,Y 524.97,Z 958.448,A -85,B 0,C 180,E1 23523.988,E2 23523.988} C_VEL
LIN {X 0,Y 524.786,Z 959.576,A -85,B 0,C 180,E1 23523.918,E2 23523.918} C_VEL
LIN {X 0,Y 522.852,Z 966.33,A -85,B 0,C 180,E1 23523.551,E2 23523.551} C_VEL
LIN {X 0,Y 514.852,Z 983.19,A -85,B 0,C 180,E1 23522.724,E2 23522.724} C_VEL
LIN {X 0,Y 512.753,Z 989.461,A -85,B 0,C 180,E1 23522.273,E2 23522.273} C_VEL
LIN {X 0,Y 509.053,Z 1007.613,A -85,B 0,C 180,E1 23520.646,E2 23520.646} C_VEL
LIN {X 0,Y 505.461,Z 1024.849,A -85,B 0,C 180,E1 23518.86,E2 23518.86} C_VEL
LIN {X 0,Y 502.16,Z 1040.194,A -85,B 0,C 180,E1 23517,E2 23517} C_VEL
LIN {X 0,Y 498.929,Z 1055.356,A -85,B 0,C 180,E1 23514.889,E2 23514.889} C_VEL
LIN {X 0,Y 496.204,Z 1068.396,A -85,B 0,C 180,E1 23512.762,E2 23512.762} C_VEL
LIN {X 0,Y 493.628,Z 1081.553,A -85,B 0,C 180,E1 23510.266,E2 23510.266} C_VEL
LIN {X 0,Y 491.708,Z 1092.155,A -85,B 0,C 180,E1 23507.882,E2 23507.882} C_VEL
LIN {X 0,Y 490.109,Z 1102.341,A -85,B 0,C 180,E1 23505.138,E2 23505.138} C_VEL
LIN {X 0,Y 489.129,Z 1109.976,A -85,B 0,C 180,E1 23502.635,E2 23502.635} C_VEL
LIN {X 0,Y 488.471,Z 1116.548,A -85,B 0,C 180,E1 23499.901,E2 23499.901} C_VEL
LIN {X 0,Y 488.147,Z 1121.138,A -85,B 0,C 180,E1 23497.414,E2 23497.414} C_VEL
LIN {X 0,Y 487.98,Z 1124.567,A -85,B 0,C 180,E1 23494.701,E2 23494.701} C_VEL
LIN {X 0,Y 487.942,Z 1126.377,A -85,B 0,C 180,E1 23492.231,E2 23492.231} C_VEL
LIN {X 0,Y 487.928,Z 1126.88,A -85,B 0,C 180,E1 23489.413,E2 23489.413} C_VEL
LIN {X 0,Y 487.946,Z 1125.971,A -85,B 0,C 180,E1 23486.946,E2 23486.946} C_VEL
LIN {X 0,Y 488.027,Z 1123.384,A -85,B 0,C 180,E1 23484.12,E2 23484.12} C_VEL
LIN {X 0,Y 488.225,Z 1119.702,A -85,B 0,C 180,E1 23481.639,E2 23481.639} C_VEL
LIN {X 0,Y 488.719,Z 1113.839,A -85,B 0,C 180,E1 23478.792,E2 23478.792} C_VEL
LIN {X 0,Y 489.474,Z 1107.166,A -85,B 0,C 180,E1 23476.293,E2 23476.293} C_VEL
LIN {X 0,Y 490.759,Z 1098.057,A -85,B 0,C 180,E1 23473.548,E2 23473.548} C_VEL
LIN {X 0,Y 492.445,Z 1088.033,A -85,B 0,C 180,E1 23471.042,E2 23471.042} C_VEL
LIN {X 0,Y 494.688,Z 1076.009,A -85,B 0,C 180,E1 23468.54,E2 23468.54} C_VEL
LIN {X 0,Y 497.412,Z 1062.698,A -85,B 0,C 180,E1 23466.168,E2 23466.168} C_VEL
LIN {X 0,Y 500.356,Z 1048.646,A -85,B 0,C 180,E1 23464.046,E2 23464.046} C_VEL
LIN {X 0,Y 503.827,Z 1032.548,A -85,B 0,C 180,E1 23461.943,E2 23461.943} C_VEL
LIN {X 0,Y 507.223,Z 1016.563,A -85,B 0,C 180,E1 23460.155,E2 23460.155} C_VEL
LIN {X 0,Y 511.168,Z 997.357,A -85,B 0,C 180,E1 23458.31,E2 23458.31} C_VEL
LIN {X 0,Y 514.598,Z 979.819,A -85,B 0,C 180,E1 23456.873,E2 23456.873} C_VEL
LIN {X 0,Y 518.295,Z 959.333,A -85,B 0,C 180,E1 23455.446,E2 23455.446} C_VEL
LIN {X 0,Y 521.412,Z 940.478,A -85,B 0,C 180,E1 23454.34,E2 23454.34} C_VEL
LIN {X 0,Y 524.656,Z 917.882,A -85,B 0,C 180,E1 23453.243,E2 23453.243} C_VEL
LIN {X 0,Y 527.101,Z 898.019,A -85,B 0,C 180,E1 23452.461,E2 23452.461} C_VEL
LIN {X 0,Y 529.441,Z 874.172,A -85,B 0,C 180,E1 23451.729,E2 23451.729} C_VEL
LIN {X 0,Y 531.121,Z 851.726,A -85,B 0,C 180,E1 23451.225,E2 23451.225} C_VEL
LIN {X 0,Y 532.49,Z 814.731,A -85,B 0,C 180,E1 23450.671,E2 23450.671} C_VEL
LIN {X 0,Y 540.587,Z 553.357,A -85,B 0,C 180,E1 23446.988,E2 23446.988} C_VEL
LIN {X 0,Y 535.188,Z 524.409,A -85,B 0,C 180,E1 23445.881,E2 23445.881} C_VEL
LIN {X 0,Y 524.68,Z 506.686,A -85,B 0,C 180,E1 23444.341,E2 23444.341} C_VEL
LIN {X 0,Y 513.826,Z 489.312,A -85,B 0,C 180,E1 23442.625,E2 23442.625} C_VEL
LIN {X 0,Y 506.968,Z 472.728,A -85,B 0,C 180,E1 23439.718,E2 23439.718} C_VEL
LIN {X 0,Y 500.098,Z 457.536,A -85,B 0,C 180,E1 23436.702,E2 23436.702} C_VEL
LIN {X 0,Y 494.17,Z 445.118,A -85,B 0,C 180,E1 23433.944,E2 23433.944} C_VEL
LIN {X 0,Y 492.395,Z 441.694,A -85,B 0,C 180,E1 23433.11,E2 23433.11} C_VEL
LIN {X 0,Y 489.95,Z 436.544,A -85,B 0,C 180,E1 23431.822,E2 23431.822} C_VEL
LIN {X 0,Y 489.939,Z 436.192,A -85,B 0,C 180,E1 23430.407,E2 23430.407} C_VEL
LIN {X 0,Y 489.914,Z 436.194,A -85,B 0,C 180,E1 23427.074,E2 23427.074} C_VEL
LIN {X 0,Y 489.897,Z 436.194,A -85,B 0,C 180,E1 23423.581,E2 23423.581} C_VEL
LIN {X 0,Y 489.933,Z 436.182,A -85,B 0,C 180,E1 23420.148,E2 23420.148} C_VEL
LIN {X 0,Y 489.939,Z 436.176,A -85,B 0,C 180,E1 23416.724,E2 23416.724} C_VEL
LIN {X 0,Y 489.907,Z 436.185,A -85,B 0,C 180,E1 23413.334,E2 23413.334} C_VEL
LIN {X 0,Y 489.937,Z 436.198,A -85,B 0,C 180,E1 23409.871,E2 23409.871} C_VEL
LIN {X 0,Y 489.976,Z 436.192,A -85,B 0,C 180,E1 23406.372,E2 23406.372} C_VEL
LIN {X 0,Y 489.925,Z 436.178,A -85,B 0,C 180,E1 23402.925,E2 23402.925} C_VEL
LIN {X 0,Y 489.925,Z 436.174,A -85,B 0,C 180,E1 23399.298,E2 23399.298} C_VEL
LIN {X 0,Y 489.974,Z 436.186,A -85,B 0,C 180,E1 23395.904,E2 23395.904} C_VEL
LIN {X 0,Y 489.954,Z 436.2,A -85,B 0,C 180,E1 23392.495,E2 23392.495} C_VEL
LIN {X 0,Y 489.937,Z 436.188,A -85,B 0,C 180,E1 23388.94,E2 23388.94} C_VEL
LIN {X 0,Y 489.963,Z 436.173,A -85,B 0,C 180,E1 23385.463,E2 23385.463} C_VEL
LIN {X 0,Y 489.988,Z 436.169,A -85,B 0,C 180,E1 23381.979,E2 23381.979} C_VEL
LIN {X 0,Y 489.957,Z 436.178,A -85,B 0,C 180,E1 23378.448,E2 23378.448} C_VEL
LIN {X 0,Y 489.954,Z 436.182,A -85,B 0,C 180,E1 23374.882,E2 23374.882} C_VEL
LIN {X 0,Y 489.989,Z 436.178,A -85,B 0,C 180,E1 23371.34,E2 23371.34} C_VEL
LIN {X 0,Y 490.001,Z 436.402,A -85,B 0,C 180,E1 23369.054,E2 23369.054} C_VEL
LIN {X 0,Y 491.434,Z 439.869,A -85,B 0,C 180,E1 23368.199,E2 23368.199} C_VEL
LIN {X 0,Y 492.535,Z 441.67,A -85,B 0,C 180,E1 23367.73,E2 23367.73} C_VEL
LIN {X 0,Y 497.265,Z 451.346,A -85,B 0,C 180,E1 23365.53,E2 23365.53} C_VEL
LIN {X 0,Y 501.736,Z 460.696,A -85,B 0,C 180,E1 23363.568,E2 23363.568} C_VEL
LIN {X 0,Y 503.309,Z 463.611,A -85,B 0,C 180,E1 23363.026,E2 23363.026} C_VEL
LIN {X 0,Y 516.362,Z 481.869,A -85,B 0,C 180,E1 23360.856,E2 23360.856} C_VEL
LIN {X 0,Y 529.014,Z 500.643,A -85,B 0,C 180,E1 23358.925,E2 23358.925} C_VEL
LIN {X 0,Y 542.619,Z 522.904,A -85,B 0,C 180,E1 23356.979,E2 23356.979} C_VEL
LIN {X 0,Y 543.466,Z 524.934,A -85,B 0,C 180,E1 23356.851,E2 23356.851} C_VEL
LIN {X 0,Y 534.752,Z 764.194,A -85,B 0,C 180,E1 23353.275,E2 23353.275} C_VEL
LIN {X 0,Y 531.786,Z 844.385,A -85,B 0,C 180,E1 23352.051,E2 23352.051} C_VEL
LIN {X 0,Y 529.917,Z 869.558,A -85,B 0,C 180,E1 23351.499,E2 23351.499} C_VEL
LIN {X 0,Y 527.739,Z 892.18,A -85,B 0,C 180,E1 23350.833,E2 23350.833} C_VEL
LIN {X 0,Y 524.951,Z 915.874,A -85,B 0,C 180,E1 23349.934,E2 23349.934} C_VEL
LIN {X 0,Y 522.141,Z 936.661,A -85,B 0,C 180,E1 23348.969,E2 23348.969} C_VEL
LIN {X 0,Y 518.59,Z 959.842,A -85,B 0,C 180,E1 23347.677,E2 23347.677} C_VEL
LIN {X 0,Y 515.401,Z 978.957,A -85,B 0,C 180,E1 23346.416,E2 23346.416} C_VEL
LIN {X 0,Y 511.623,Z 1000.122,A -85,B 0,C 180,E1 23344.797,E2 23344.797} C_VEL
LIN {X 0,Y 508.153,Z 1018.435,A -85,B 0,C 180,E1 23343.163,E2 23343.163} C_VEL
LIN {X 0,Y 504.536,Z 1037.382,A -85,B 0,C 180,E1 23341.226,E2 23341.226} C_VEL
LIN {X 0,Y 501.227,Z 1054.473,A -85,B 0,C 180,E1 23339.193,E2 23339.193} C_VEL
LIN {X 0,Y 498.122,Z 1070.894,A -85,B 0,C 180,E1 23336.969,E2 23336.969} C_VEL
LIN {X 0,Y 495.485,Z 1085.343,A -85,B 0,C 180,E1 23334.691,E2 23334.691} C_VEL
LIN {X 0,Y 493.125,Z 1099.409,A -85,B 0,C 180,E1 23332.157,E2 23332.157} C_VEL
LIN {X 0,Y 491.292,Z 1111.331,A -85,B 0,C 180,E1 23329.622,E2 23329.622} C_VEL
LIN {X 0,Y 489.914,Z 1122.104,A -85,B 0,C 180,E1 23326.969,E2 23326.969} C_VEL
LIN {X 0,Y 488.963,Z 1130.919,A -85,B 0,C 180,E1 23324.326,E2 23324.326} C_VEL
LIN {X 0,Y 488.402,Z 1137.921,A -85,B 0,C 180,E1 23321.814,E2 23321.814} C_VEL
LIN {X 0,Y 488.065,Z 1144.123,A -85,B 0,C 180,E1 23318.957,E2 23318.957} C_VEL
LIN {X 0,Y 487.962,Z 1147.958,A -85,B 0,C 180,E1 23316.589,E2 23316.589} C_VEL
LIN {X 0,Y 487.929,Z 1150.999,A -85,B 0,C 180,E1 23313.878,E2 23313.878} C_VEL
LIN {X 0,Y 487.928,Z 1152.339,A -85,B 0,C 180,E1 23311.174,E2 23311.174} C_VEL
LIN {X 0,Y 487.923,Z 1152.362,A -85,B 0,C 180,E1 23308.943,E2 23308.943} C_VEL
LIN {X 0,Y 487.926,Z 1151.154,A -85,B 0,C 180,E1 23306.358,E2 23306.358} C_VEL
LIN {X 0,Y 487.96,Z 1148.121,A -85,B 0,C 180,E1 23303.529,E2 23303.529} C_VEL
LIN {X 0,Y 488.059,Z 1144.335,A -85,B 0,C 180,E1 23301.161,E2 23301.161} C_VEL
LIN {X 0,Y 488.362,Z 1138.543,A -85,B 0,C 180,E1 23298.425,E2 23298.425} C_VEL
LIN {X 0,Y 488.933,Z 1131.232,A -85,B 0,C 180,E1 23295.779,E2 23295.779} C_VEL
LIN {X 0,Y 489.837,Z 1122.717,A -85,B 0,C 180,E1 23293.208,E2 23293.208} C_VEL
LIN {X 0,Y 491.218,Z 1111.856,A -85,B 0,C 180,E1 23290.499,E2 23290.499} C_VEL
LIN {X 0,Y 492.931,Z 1100.58,A -85,B 0,C 180,E1 23288.085,E2 23288.085} C_VEL
LIN {X 0,Y 495.234,Z 1086.762,A -85,B 0,C 180,E1 23285.55,E2 23285.55} C_VEL
LIN {X 0,Y 497.672,Z 1073.178,A -85,B 0,C 180,E1 23283.382,E2 23283.382} C_VEL
LIN {X 0,Y 501.02,Z 1055.508,A -85,B 0,C 180,E1 23280.942,E2 23280.942} C_VEL
LIN {X 0,Y 504.099,Z 1039.502,A -85,B 0,C 180,E1 23279.021,E2 23279.021} C_VEL
LIN {X 0,Y 507.91,Z 1019.617,A -85,B 0,C 180,E1 23276.954,E2 23276.954} C_VEL
LIN {X 0,Y 511.349,Z 1001.408,A -85,B 0,C 180,E1 23275.318,E2 23275.318} C_VEL
LIN {X 0,Y 515.24,Z 979.764,A -85,B 0,C 180,E1 23273.646,E2 23273.646} C_VEL
LIN {X 0,Y 518.441,Z 960.583,A -85,B 0,C 180,E1 23272.374,E2 23272.374} C_VEL
LIN {X 0,Y 521.998,Z 937.466,A -85,B 0,C 180,E1 23271.076,E2 23271.076} C_VEL
LIN {X 0,Y 524.808,Z 916.719,A -85,B 0,C 180,E1 23270.108,E2 23270.108} C_VEL
LIN {X 0,Y 527.668,Z 892.544,A -85,B 0,C 180,E1 23269.184,E2 23269.184} C_VEL
LIN {X 0,Y 529.856,Z 869.812,A -85,B 0,C 180,E1 23268.513,E2 23268.513} C_VEL
LIN {X 0,Y 531.733,Z 844.621,A -85,B 0,C 180,E1 23267.958,E2 23267.958} C_VEL
LIN {X 0,Y 534.605,Z 767.134,A -85,B 0,C 180,E1 23266.775,E2 23266.775} C_VEL
LIN {X 0,Y 543.258,Z 528.876,A -85,B 0,C 180,E1 23263.213,E2 23263.213} C_VEL
LIN {X 0,Y 543.32,Z 524.225,A -85,B 0,C 180,E1 23263.132,E2 23263.132} C_VEL
LIN {X 0,Y 531.17,Z 504.172,A -85,B 0,C 180,E1 23261.41,E2 23261.41} C_VEL
LIN {X 0,Y 518.452,Z 484.878,A -85,B 0,C 180,E1 23259.491,E2 23259.491} C_VEL
LIN {X 0,Y 505.655,Z 466.879,A -85,B 0,C 180,E1 23257.414,E2 23257.414} C_VEL
LIN {X 0,Y 502.921,Z 462.905,A -85,B 0,C 180,E1 23256.901,E2 23256.901} C_VEL
LIN {X 0,Y 496.57,Z 449.64,A -85,B 0,C 180,E1 23254.148,E2 23254.148} C_VEL
LIN {X 0,Y 491.657,Z 440.163,A -85,B 0,C 180,E1 23251.922,E2 23251.922} C_VEL
LIN {X 0,Y 490.05,Z 436.72,A -85,B 0,C 180,E1 23251.079,E2 23251.079} C_VEL
LIN {X 0,Y 489.994,Z 436.204,A -85,B 0,C 180,E1 23250.674,E2 23250.674} C_VEL
LIN {X 0,Y 489.96,Z 436.194,A -85,B 0,C 180,E1 23247.155,E2 23247.155} C_VEL
LIN {X 0,Y 489.96,Z 436.193,A -85,B 0,C 180,E1 23243.578,E2 23243.578} C_VEL
LIN {X 0,Y 489.995,Z 436.196,A -85,B 0,C 180,E1 23240.168,E2 23240.168} C_VEL
LIN {X 0,Y 489.966,Z 436.195,A -85,B 0,C 180,E1 23236.601,E2 23236.601} C_VEL
LIN {X 0,Y 489.94,Z 436.185,A -85,B 0,C 180,E1 23233.093,E2 23233.093} C_VEL
LIN {X 0,Y 489.965,Z 436.172,A -85,B 0,C 180,E1 23229.633,E2 23229.633} C_VEL
LIN {X 0,Y 489.974,Z 436.176,A -85,B 0,C 180,E1 23226.209,E2 23226.209} C_VEL
LIN {X 0,Y 489.935,Z 436.201,A -85,B 0,C 180,E1 23222.69,E2 23222.69} C_VEL
LIN {X 0,Y 489.934,Z 436.199,A -85,B 0,C 180,E1 23219.064,E2 23219.064} C_VEL
LIN {X 0,Y 489.967,Z 436.173,A -85,B 0,C 180,E1 23215.552,E2 23215.552} C_VEL
LIN {X 0,Y 489.934,Z 436.175,A -85,B 0,C 180,E1 23212.259,E2 23212.259} C_VEL
LIN {X 0,Y 489.918,Z 436.193,A -85,B 0,C 180,E1 23208.701,E2 23208.701} C_VEL
LIN {X 0,Y 489.945,Z 436.203,A -85,B 0,C 180,E1 23205.22,E2 23205.22} C_VEL
LIN {X 0,Y 489.948,Z 436.192,A -85,B 0,C 180,E1 23201.805,E2 23201.805} C_VEL
LIN {X 0,Y 489.902,Z 436.186,A -85,B 0,C 180,E1 23198.446,E2 23198.446} C_VEL
LIN {X 0,Y 489.929,Z 436.181,A -85,B 0,C 180,E1 23195.01,E2 23195.01} C_VEL
LIN {X 0,Y 489.941,Z 436.18,A -85,B 0,C 180,E1 23191.595,E2 23191.595} C_VEL
LIN {X 0,Y 489.903,Z 436.276,A -85,B 0,C 180,E1 23188.225,E2 23188.225} C_VEL
LIN {X 0,Y 490.028,Z 436.932,A -85,B 0,C 180,E1 23187.959,E2 23187.959} C_VEL
LIN {X 0,Y 491.981,Z 440.663,A -85,B 0,C 180,E1 23186.997,E2 23186.997} C_VEL
LIN {X 0,Y 493.903,Z 444.771,A -85,B 0,C 180,E1 23186.03,E2 23186.03} C_VEL
LIN {X 0,Y 498.996,Z 455.304,A -85,B 0,C 180,E1 23183.662,E2 23183.662} C_VEL
LIN {X 0,Y 504.201,Z 466.656,A -85,B 0,C 180,E1 23181.341,E2 23181.341} C_VEL
LIN {X 0,Y 510.4,Z 480.952,A -85,B 0,C 180,E1 23178.685,E2 23178.685} C_VEL
LIN {X 0,Y 514.182,Z 490.02,A -85,B 0,C 180,E1 23177.184,E2 23177.184} C_VEL
LIN {X 0,Y 526.197,Z 509.214,A -85,B 0,C 180,E1 23175.325,E2 23175.325} C_VEL
LIN {X 0,Y 535.402,Z 525.1,A -85,B 0,C 180,E1 23173.979,E2 23173.979} C_VEL
LIN {X 0,Y 540.503,Z 554.048,A -85,B 0,C 180,E1 23172.907,E2 23172.907} C_VEL
LIN {X 0,Y 532.417,Z 815.635,A -85,B 0,C 180,E1 23169.221,E2 23169.221} C_VEL
LIN {X 0,Y 531.065,Z 851.885,A -85,B 0,C 180,E1 23168.676,E2 23168.676} C_VEL
LIN {X 0,Y 529.399,Z 874.159,A -85,B 0,C 180,E1 23168.175,E2 23168.175} C_VEL
LIN {X 0,Y 527.073,Z 897.952,A -85,B 0,C 180,E1 23167.446,E2 23167.446} C_VEL
LIN {X 0,Y 524.694,Z 917.306,A -85,B 0,C 180,E1 23166.686,E2 23166.686} C_VEL
LIN {X 0,Y 521.548,Z 939.433,A -85,B 0,C 180,E1 23165.622,E2 23165.622} C_VEL
LIN {X 0,Y 518.331,Z 958.92,A -85,B 0,C 180,E1 23164.484,E2 23164.484} C_VEL
LIN {X 0,Y 514.418,Z 980.566,A -85,B 0,C 180,E1 23162.973,E2 23162.973} C_VEL
LIN {X 0,Y 512.753,Z 989.461,A -85,B 0,C 180,E1 23162.273,E2 23162.273} C_VEL
LIN {X 0,Y 510.628,Z 995.695,A -85,B 0,C 180,E1 23161.802,E2 23161.802} C_VEL
LIN {X 0,Y 502.258,Z 1011.324,A -85,B 0,C 180,E1 23160.728,E2 23160.728} C_VEL
LIN {X 0,Y 500.137,Z 1017.069,A -85,B 0,C 180,E1 23160.192,E2 23160.192} C_VEL
LIN {X 0,Y 496.589,Z 1033.145,A -85,B 0,C 180,E1 23158.368,E2 23158.368} C_VEL
LIN {X 0,Y 492.973,Z 1049.143,A -85,B 0,C 180,E1 23156.242,E2 23156.242} C_VEL
LIN {X 0,Y 489.755,Z 1063.885,A -85,B 0,C 180,E1 23153.972,E2 23153.972} C_VEL
LIN {X 0,Y 487.058,Z 1076.423,A -85,B 0,C 180,E1 23151.686,E2 23151.686} C_VEL
LIN {X 0,Y 484.705,Z 1088.405,A -85,B 0,C 180,E1 23149.147,E2 23149.147} C_VEL
LIN {X 0,Y 483.005,Z 1097.959,A -85,B 0,C 180,E1 23146.723,E2 23146.723} C_VEL
LIN {X 0,Y 481.626,Z 1107.132,A -85,B 0,C 180,E1 23143.935,E2 23143.935} C_VEL
LIN {X 0,Y 480.804,Z 1113.837,A -85,B 0,C 180,E1 23141.395,E2 23141.395} C_VEL
LIN {X 0,Y 480.27,Z 1119.765,A -85,B 0,C 180,E1 23138.501,E2 23138.501} C_VEL
LIN {X 0,Y 480.04,Z 1123.477,A -85,B 0,C 180,E1 23135.978,E2 23135.978} C_VEL
LIN {X 0,Y 479.953,Z 1126.13,A -85,B 0,C 180,E1 23133.105,E2 23133.105} C_VEL
LIN {X 0,Y 479.936,Z 1127.073,A -85,B 0,C 180,E1 23130.597,E2 23130.597} C_VEL
LIN {X 0,Y 479.942,Z 1126.64,A -85,B 0,C 180,E1 23127.731,E2 23127.731} C_VEL
LIN {X 0,Y 479.983,Z 1124.867,A -85,B 0,C 180,E1 23125.22,E2 23125.22} C_VEL
LIN {X 0,Y 480.164,Z 1121.418,A -85,B 0,C 180,E1 23122.404,E2 23122.404} C_VEL
LIN {X 0,Y 480.516,Z 1116.716,A -85,B 0,C 180,E1 23119.812,E2 23119.812} C_VEL
LIN {X 0,Y 481.268,Z 1109.79,A -85,B 0,C 180,E1 23116.911,E2 23116.911} C_VEL
LIN {X 0,Y 482.282,Z 1102.487,A -85,B 0,C 180,E1 23114.487,E2 23114.487} C_VEL
LIN {X 0,Y 483.988,Z 1092.282,A -85,B 0,C 180,E1 23111.698,E2 23111.698} C_VEL
LIN {X 0,Y 486.014,Z 1081.671,A -85,B 0,C 180,E1 23109.276,E2 23109.276} C_VEL
LIN {X 0,Y 488.737,Z 1068.499,A -85,B 0,C 180,E1 23106.743,E2 23106.743} C_VEL
LIN {X 0,Y 491.789,Z 1054.696,A -85,B 0,C 180,E1 23104.467,E2 23104.467} C_VEL
LIN {X 0,Y 495.19,Z 1039.359,A -85,B 0,C 180,E1 23102.327,E2 23102.327} C_VEL
LIN {X 0,Y 498.908,Z 1022.825,A -85,B 0,C 180,E1 23100.328,E2 23100.328} C_VEL
LIN {X 0,Y 502.588,Z 1005.866,A -85,B 0,C 180,E1 23098.584,E2 23098.584} C_VEL
LIN {X 0,Y 506.513,Z 987.099,A -85,B 0,C 180,E1 23096.918,E2 23096.918} C_VEL
LIN {X 0,Y 510.151,Z 968.188,A -85,B 0,C 180,E1 23095.498,E2 23095.498} C_VEL
LIN {X 0,Y 514.086,Z 945.955,A -85,B 0,C 180,E1 23094.097,E2 23094.097} C_VEL
LIN {X 0,Y 517.085,Z 926.908,A -85,B 0,C 180,E1 23093.1,E2 23093.1} C_VEL
LIN {X 0,Y 520.12,Z 904.488,A -85,B 0,C 180,E1 23092.14,E2 23092.14} C_VEL
LIN {X 0,Y 522.393,Z 884.201,A -85,B 0,C 180,E1 23091.449,E2 23091.449} C_VEL
LIN {X 0,Y 524.477,Z 860.054,A -85,B 0,C 180,E1 23090.829,E2 23090.829} C_VEL
LIN {X 0,Y 525.719,Z 838.008,A -85,B 0,C 180,E1 23090.431,E2 23090.431} C_VEL
LIN {X 0,Y 533.698,Z 588.129,A -85,B 0,C 180,E1 23086.878,E2 23086.878} C_VEL
LIN {X 0,Y 534.725,Z 554.099,A -85,B 0,C 180,E1 23086.373,E2 23086.373} C_VEL
LIN {X 0,Y 530.06,Z 528.816,A -85,B 0,C 180,E1 23085.388,E2 23085.388} C_VEL
LIN {X 0,Y 520.334,Z 512.241,A -85,B 0,C 180,E1 23083.925,E2 23083.925} C_VEL
LIN {X 0,Y 508.624,Z 493.694,A -85,B 0,C 180,E1 23082.057,E2 23082.057} C_VEL
LIN {X 0,Y 505.505,Z 488.711,A -85,B 0,C 180,E1 23081.501,E2 23081.501} C_VEL
LIN {X 0,Y 499.314,Z 474.115,A -85,B 0,C 180,E1 23078.814,E2 23078.814} C_VEL
LIN {X 0,Y 493.683,Z 461.638,A -85,B 0,C 180,E1 23076.257,E2 23076.257} C_VEL
LIN {X 0,Y 488.616,Z 450.786,A -85,B 0,C 180,E1 23073.816,E2 23073.816} C_VEL
LIN {X 0,Y 485.565,Z 445.07,A -85,B 0,C 180,E1 23072.371,E2 23072.371} C_VEL
LIN {X 0,Y 483.696,Z 441.24,A -85,B 0,C 180,E1 23071.395,E2 23071.395} C_VEL
LIN {X 0,Y 482.009,Z 437.334,A -85,B 0,C 180,E1 23070.305,E2 23070.305} C_VEL
LIN {X 0,Y 481.98,Z 437.183,A -85,B 0,C 180,E1 23067.022,E2 23067.022} C_VEL
LIN {X 0,Y 481.959,Z 437.183,A -85,B 0,C 180,E1 23063.509,E2 23063.509} C_VEL
LIN {X 0,Y 481.981,Z 437.174,A -85,B 0,C 180,E1 23059.986,E2 23059.986} C_VEL
LIN {X 0,Y 482.02,Z 437.162,A -85,B 0,C 180,E1 23056.51,E2 23056.51} C_VEL
LIN {X 0,Y 481.97,Z 437.171,A -85,B 0,C 180,E1 23053.191,E2 23053.191} C_VEL
LIN {X 0,Y 481.978,Z 437.182,A -85,B 0,C 180,E1 23049.553,E2 23049.553} C_VEL
LIN {X 0,Y 482.041,Z 437.184,A -85,B 0,C 180,E1 23046.192,E2 23046.192} C_VEL
LIN {X 0,Y 482.005,Z 437.169,A -85,B 0,C 180,E1 23042.616,E2 23042.616} C_VEL
LIN {X 0,Y 481.984,Z 437.162,A -85,B 0,C 180,E1 23039.168,E2 23039.168} C_VEL
LIN {X 0,Y 482.018,Z 437.171,A -85,B 0,C 180,E1 23035.717,E2 23035.717} C_VEL
LIN {X 0,Y 482.039,Z 437.188,A -85,B 0,C 180,E1 23032.251,E2 23032.251} C_VEL
LIN {X 0,Y 482.003,Z 437.179,A -85,B 0,C 180,E1 23028.755,E2 23028.755} C_VEL
LIN {X 0,Y 482.003,Z 437.167,A -85,B 0,C 180,E1 23025.094,E2 23025.094} C_VEL
LIN {X 0,Y 482.044,Z 437.157,A -85,B 0,C 180,E1 23021.622,E2 23021.622} C_VEL
LIN {X 0,Y 482.052,Z 437.159,A -85,B 0,C 180,E1 23018.001,E2 23018.001} C_VEL
LIN {X 0,Y 482.018,Z 437.166,A -85,B 0,C 180,E1 23014.439,E2 23014.439} C_VEL
LIN {X 0,Y 482.022,Z 437.182,A -85,B 0,C 180,E1 23010.825,E2 23010.825} C_VEL
LIN {X 0,Y 482.105,Z 437.693,A -85,B 0,C 180,E1 23010.378,E2 23010.378} C_VEL
LIN {X 0,Y 483.797,Z 441.25,A -85,B 0,C 180,E1 23009.441,E2 23009.441} C_VEL
LIN {X 0,Y 484.751,Z 443.151,A -85,B 0,C 180,E1 23008.957,E2 23008.957} C_VEL
LIN {X 0,Y 487.24,Z 447.981,A -85,B 0,C 180,E1 23007.754,E2 23007.754} C_VEL
LIN {X 0,Y 491.387,Z 456.191,A -85,B 0,C 180,E1 23005.832,E2 23005.832} C_VEL
LIN {X 0,Y 495.3,Z 464.041,A -85,B 0,C 180,E1 23004.184,E2 23004.184} C_VEL
LIN {X 0,Y 508.955,Z 482.863,A -85,B 0,C 180,E1 23001.804,E2 23001.804} C_VEL
LIN {X 0,Y 522.678,Z 503.241,A -85,B 0,C 180,E1 22999.624,E2 22999.624} C_VEL
LIN {X 0,Y 535.96,Z 524.785,A -85,B 0,C 180,E1 22997.663,E2 22997.663} C_VEL
LIN {X 0,Y 537.701,Z 528.15,A -85,B 0,C 180,E1 22997.408,E2 22997.408} C_VEL
LIN {X 0,Y 528.716,Z 765.855,A -85,B 0,C 180,E1 22993.826,E2 22993.826} C_VEL
LIN {X 0,Y 525.697,Z 844.488,A -85,B 0,C 180,E1 22992.615,E2 22992.615} C_VEL
LIN {X 0,Y 523.762,Z 869.697,A -85,B 0,C 180,E1 22992.057,E2 22992.057} C_VEL
LIN {X 0,Y 521.493,Z 892.462,A -85,B 0,C 180,E1 22991.382,E2 22991.382} C_VEL
LIN {X 0,Y 518.592,Z 916.173,A -85,B 0,C 180,E1 22990.472,E2 22990.472} C_VEL
LIN {X 0,Y 515.653,Z 937.148,A -85,B 0,C 180,E1 22989.488,E2 22989.488} C_VEL
LIN {X 0,Y 511.955,Z 960.284,A -85,B 0,C 180,E1 22988.181,E2 22988.181} C_VEL
LIN {X 0,Y 508.652,Z 979.345,A -85,B 0,C 180,E1 22986.909,E2 22986.909} C_VEL
LIN {X 0,Y 504.591,Z 1001.1,A -85,B 0,C 180,E1 22985.215,E2 22985.215} C_VEL
LIN {X 0,Y 501.124,Z 1018.694,A -85,B 0,C 180,E1 22983.621,E2 22983.621} C_VEL
LIN {X 0,Y 497.218,Z 1038.18,A -85,B 0,C 180,E1 22981.592,E2 22981.592} C_VEL
LIN {X 0,Y 493.893,Z 1054.631,A -85,B 0,C 180,E1 22979.603,E2 22979.603} C_VEL
LIN {X 0,Y 490.574,Z 1071.346,A -85,B 0,C 180,E1 22977.294,E2 22977.294} C_VEL
LIN {X 0,Y 487.916,Z 1085.236,A -85,B 0,C 180,E1 22975.069,E2 22975.069} C_VEL
LIN {X 0,Y 485.454,Z 1099.143,A -85,B 0,C 180,E1 22972.526,E2 22972.526} C_VEL
LIN {X 0,Y 483.52,Z 1111.072,A -85,B 0,C 180,E1 22969.951,E2 22969.951} C_VEL
LIN {X 0,Y 482.051,Z 1121.857,A -85,B 0,C 180,E1 22967.255,E2 22967.255} C_VEL
LIN {X 0,Y 481.038,Z 1130.679,A -85,B 0,C 180,E1 22964.567,E2 22964.567} C_VEL
LIN {X 0,Y 480.438,Z 1137.737,A -85,B 0,C 180,E1 22961.993,E2 22961.993} C_VEL
LIN {X 0,Y 480.075,Z 1143.901,A -85,B 0,C 180,E1 22959.108,E2 22959.108} C_VEL
LIN {X 0,Y 479.966,Z 1147.74,A -85,B 0,C 180,E1 22956.7,E2 22956.7} C_VEL
LIN {X 0,Y 479.931,Z 1150.786,A -85,B 0,C 180,E1 22953.942,E2 22953.942} C_VEL
LIN {X 0,Y 479.93,Z 1152.129,A -85,B 0,C 180,E1 22951.194,E2 22951.194} C_VEL
LIN {X 0,Y 479.927,Z 1152.152,A -85,B 0,C 180,E1 22948.926,E2 22948.926} C_VEL
LIN {X 0,Y 479.929,Z 1150.968,A -85,B 0,C 180,E1 22946.34,E2 22946.34} C_VEL
LIN {X 0,Y 479.961,Z 1148.069,A -85,B 0,C 180,E1 22943.541,E2 22943.541} C_VEL
LIN {X 0,Y 480.06,Z 1144.326,A -85,B 0,C 180,E1 22941.134,E2 22941.134} C_VEL
LIN {X 0,Y 480.375,Z 1138.615,A -85,B 0,C 180,E1 22938.352,E2 22938.352} C_VEL
LIN {X 0,Y 480.975,Z 1131.296,A -85,B 0,C 180,E1 22935.642,E2 22935.642} C_VEL
LIN {X 0,Y 481.833,Z 1123.524,A -85,B 0,C 180,E1 22933.235,E2 22933.235} C_VEL
LIN {X 0,Y 483.36,Z 1112.124,A -85,B 0,C 180,E1 22930.294,E2 22930.294} C_VEL
LIN {X 0,Y 485.146,Z 1100.9,A -85,B 0,C 180,E1 22927.842,E2 22927.842} C_VEL
LIN {X 0,Y 487.686,Z 1086.475,A -85,B 0,C 180,E1 22925.146,E2 22925.146} C_VEL
LIN {X 0,Y 490.252,Z 1072.881,A -85,B 0,C 180,E1 22922.947,E2 22922.947} C_VEL
LIN {X 0,Y 493.703,Z 1055.539,A -85,B 0,C 180,E1 22920.518,E2 22920.518} C_VEL
LIN {X 0,Y 496.89,Z 1039.686,A -85,B 0,C 180,E1 22918.588,E2 22918.588} C_VEL
LIN {X 0,Y 500.87,Z 1019.868,A -85,B 0,C 180,E1 22916.497,E2 22916.497} C_VEL
LIN {X 0,Y 504.386,Z 1001.987,A -85,B 0,C 180,E1 22914.868,E2 22914.868} C_VEL
LIN {X 0,Y 508.497,Z 980.068,A -85,B 0,C 180,E1 22913.148,E2 22913.148} C_VEL
LIN {X 0,Y 511.789,Z 961.089,A -85,B 0,C 180,E1 22911.875,E2 22911.875} C_VEL
LIN {X 0,Y 515.333,Z 939.171,A -85,B 0,C 180,E1 22910.619,E2 22910.619} C_VEL
LIN {X 0,Y 518.358,Z 917.66,A -85,B 0,C 180,E1 22909.599,E2 22909.599} C_VEL
LIN {X 0,Y 521.293,Z 894.078,A -85,B 0,C 180,E1 22908.677,E2 22908.677} C_VEL
LIN {X 0,Y 523.646,Z 870.487,A -85,B 0,C 180,E1 22907.97,E2 22907.97} C_VEL
LIN {X 0,Y 525.588,Z 845.742,A -85,B 0,C 180,E1 22907.412,E2 22907.412} C_VEL
LIN {X 0,Y 528.028,Z 783.566,A -85,B 0,C 180,E1 22906.448,E2 22906.448} C_VEL
LIN {X 0,Y 536.717,Z 551.678,A -85,B 0,C 180,E1 22902.949,E2 22902.949} C_VEL
LIN {X 0,Y 537.554,Z 527.604,A -85,B 0,C 180,E1 22902.579,E2 22902.579} C_VEL
LIN {X 0,Y 524.368,Z 505.898,A -85,B 0,C 180,E1 22900.65,E2 22900.65} C_VEL
LIN {X 0,Y 511.133,Z 486.015,A -85,B 0,C 180,E1 22898.576,E2 22898.576} C_VEL
LIN {X 0,Y 498.308,Z 468.273,A -85,B 0,C 180,E1 22896.402,E2 22896.402} C_VEL
LIN {X 0,Y 494.851,Z 463.376,A -85,B 0,C 180,E1 22895.729,E2 22895.729} C_VEL
LIN {X 0,Y 490.161,Z 453.905,A -85,B 0,C 180,E1 22893.665,E2 22893.665} C_VEL
LIN {X 0,Y 486.179,Z 445.874,A -85,B 0,C 180,E1 22891.769,E2 22891.769} C_VEL
LIN {X 0,Y 483.711,Z 441.142,A -85,B 0,C 180,E1 22890.565,E2 22890.565} C_VEL
LIN {X 0,Y 482.048,Z 437.358,A -85,B 0,C 180,E1 22889.551,E2 22889.551} C_VEL
LIN {X 0,Y 482.05,Z 437.162,A -85,B 0,C 180,E1 22886.084,E2 22886.084} C_VEL
LIN {X 0,Y 482.043,Z 437.161,A -85,B 0,C 180,E1 22882.566,E2 22882.566} C_VEL
LIN {X 0,Y 482.011,Z 437.167,A -85,B 0,C 180,E1 22879.007,E2 22879.007} C_VEL
LIN {X 0,Y 482.012,Z 437.175,A -85,B 0,C 180,E1 22875.398,E2 22875.398} C_VEL
LIN {X 0,Y 482.045,Z 437.186,A -85,B 0,C 180,E1 22871.85,E2 22871.85} C_VEL
LIN {X 0,Y 482.039,Z 437.181,A -85,B 0,C 180,E1 22868.229,E2 22868.229} C_VEL
LIN {X 0,Y 481.996,Z 437.166,A -85,B 0,C 180,E1 22864.76,E2 22864.76} C_VEL
LIN {X 0,Y 481.998,Z 437.161,A -85,B 0,C 180,E1 22861.189,E2 22861.189} C_VEL
LIN {X 0,Y 482.04,Z 437.173,A -85,B 0,C 180,E1 22857.741,E2 22857.741} C_VEL
LIN {X 0,Y 482.009,Z 437.188,A -85,B 0,C 180,E1 22854.166,E2 22854.166} C_VEL
LIN {X 0,Y 481.979,Z 437.175,A -85,B 0,C 180,E1 22850.688,E2 22850.688} C_VEL
LIN {X 0,Y 481.998,Z 437.164,A -85,B 0,C 180,E1 22847.163,E2 22847.163} C_VEL
LIN {X 0,Y 482.012,Z 437.167,A -85,B 0,C 180,E1 22843.834,E2 22843.834} C_VEL
LIN {X 0,Y 481.971,Z 437.182,A -85,B 0,C 180,E1 22840.361,E2 22840.361} C_VEL
LIN {X 0,Y 481.977,Z 437.189,A -85,B 0,C 180,E1 22836.786,E2 22836.786} C_VEL
LIN {X 0,Y 482.016,Z 437.186,A -85,B 0,C 180,E1 22833.247,E2 22833.247} C_VEL
LIN {X 0,Y 481.973,Z 437.194,A -85,B 0,C 180,E1 22829.864,E2 22829.864} C_VEL
LIN {X 0,Y 482.105,Z 437.72,A -85,B 0,C 180,E1 22829.397,E2 22829.397} C_VEL
LIN {X 0,Y 483.707,Z 441.268,A -85,B 0,C 180,E1 22828.467,E2 22828.467} C_VEL
LIN {X 0,Y 486.849,Z 447.471,A -85,B 0,C 180,E1 22826.885,E2 22826.885} C_VEL
LIN {X 0,Y 490.905,Z 455.622,A -85,B 0,C 180,E1 22824.943,E2 22824.943} C_VEL
LIN {X 0,Y 496.922,Z 468.726,A -85,B 0,C 180,E1 22822.141,E2 22822.141} C_VEL
LIN {X 0,Y 502.712,Z 482.005,A -85,B 0,C 180,E1 22819.578,E2 22819.578} C_VEL
LIN {X 0,Y 505.882,Z 489.523,A -85,B 0,C 180,E1 22818.291,E2 22818.291} C_VEL
LIN {X 0,Y 518.383,Z 509.038,A -85,B 0,C 180,E1 22816.27,E2 22816.27} C_VEL
LIN {X 0,Y 528.97,Z 526.982,A -85,B 0,C 180,E1 22814.666,E2 22814.666} C_VEL
LIN {X 0,Y 530.324,Z 529.838,A -85,B 0,C 180,E1 22814.459,E2 22814.459} C_VEL
LIN {X 0,Y 534.782,Z 555.638,A -85,B 0,C 180,E1 22813.489,E2 22813.489} C_VEL
LIN {X 0,Y 526.378,Z 816.151,A -85,B 0,C 180,E1 22809.786,E2 22809.786} C_VEL
LIN {X 0,Y 524.99,Z 851.864,A -85,B 0,C 180,E1 22809.244,E2 22809.244} C_VEL
LIN {X 0,Y 523.258,Z 874.23,A -85,B 0,C 180,E1 22808.738,E2 22808.738} C_VEL
LIN {X 0,Y 520.859,Z 897.943,A -85,B 0,C 180,E1 22808.006,E2 22808.006} C_VEL
LIN {X 0,Y 518.313,Z 917.943,A -85,B 0,C 180,E1 22807.213,E2 22807.213} C_VEL
